METHOD PROTECTED OnExecute
hresult.Value := F_VN_MinPixelValueExp(
	ipImage := ipImage.Value,
    aMinValue := aMinValue.Value,
    aPosition := aPosition.Value,
    ipMask := ipMask.Value,
    eVectorCompareMethod := eVectorCompareMethod.Value,
	hrPrev:= hrPrev.Value);
END_METHOD

METHOD PUBLIC PreExecutionCheck
VAR_INPUT
	Check : I_PreExecutionChecks;
END_VAR
Check.IsTrue(ipImage.IsValid, 'ipImage must contain an image');
Check.IsTrue((ipImage.HasChannelCount(1) OR
              ipImage.HasChannelCount(2) OR
              ipImage.HasChannelCount(3) OR
              ipImage.HasChannelCount(4)), 'ipImage must contain 1, 2, 3 or 4 channels');

// ipMask : Optional mask to specify which pixel positions are considered (USINT, set parameter to 0 if not required)
IF NOT IsValidImage(ipMask.Value) THEN
    RETURN;
END_IF

Check.IsTrue(ipMask.IsValid, 'ipMask must contain an image');
Check.IsTrue(ipMask.HasChannelCount(1), 'ipMask must have 1 channel');
Check.IsTrue(ipMask.IsPixelDepth(8), 'ipMask must have 8 bit pixel depth');
Check.IsTrue(IsImage1SizeEqualToImage2Size(ipMask.Value, ipImage.Value), 'ipMask must be the same size as ipImage');
END_METHOD

END_FUNCTION_BLOCK

// ---- Nodes/Image Analysis/Node_F_VN_MinPixelValue.TcPOU
{attribute 'linkalways'} 
{attribute 'no_explicit_call' := 'This FB is a CLASS and must be accessed using methods or properties'}
{attribute 'enable_dynamic_creation'}
FUNCTION_BLOCK Node_F_VN_MinPixelValue EXTENDS VisionNode
VAR
    ipImage : _ITcVnImage;
    aMinValue : _TcVnVector4_LREAL;
    aPosition : _TcVnPoint2_DINT;
    hrPrev : _HRESULT(S_OK);
	hresult : _HRESULT(S_OK);
END_VAR

METHOD PUBLIC  Clone : I_Node
VAR
	pNode : POINTER TO Node_F_VN_MinPixelValue;
END_VAR
pNode := __NEW(Node_F_VN_MinPixelValue);
Clone := pNode^;
END_METHOD

METHOD FB_init : BOOL
VAR_INPUT
	bInitRetains : BOOL; // if TRUE, the retain variables are initialized (warm start / cold start)
	bInCopyCode : BOOL;  // if TRUE, the instance afterwards gets moved into the copy code (online change)
END_VAR
AddInput('ipImage', ipImage);
AddInput('hrPrev', hrPrev);
AddOutput('aMinValue', aMinValue);
AddOutput('aPosition', aPosition);
AddOutput('hresult', hresult);
END_METHOD

METHOD PROTECTED OnExecute
hresult.Value := F_VN_MinPixelValue(
	ipImage := ipImage.Value,
    aMinValue := aMinValue.Value,
    aPosition := aPosition.Value,
	hrPrev:= hrPrev.Value);
END_METHOD

METHOD PUBLIC PreExecutionCheck
VAR_INPUT
	Check : I_PreExecutionChecks;
END_VAR
Check.IsTrue(ipImage.IsValid, 'ipImage must contain an image');
Check.IsTrue((ipImage.HasChannelCount(1) OR
              ipImage.HasChannelCount(2) OR
              ipImage.HasChannelCount(3) OR
              ipImage.HasChannelCount(4)), 'ipImage must contain 1, 2, 3 or 4 channels');
END_METHOD

END_FUNCTION_BLOCK

// ---- Nodes/Image Analysis/Node_F_VN_RegionOrientationExp.TcPOU
{attribute 'linkalways'} 
{attribute 'no_explicit_call' := 'This FB is a CLASS and must be accessed using methods or properties'}
{attribute 'enable_dynamic_creation'}
FUNCTION_BLOCK Node_F_VN_RegionOrientationExp EXTENDS VisionNode
VAR
    ipSrcImage : _ITcVnImage;
    stOrientation : _TcVnRotatedRectangle;
    eMethod : _ETcVnOrientationMethod(ETcVnOrientationMethod.TCVN_OM_PCA);
    hrPrev : _HRESULT(S_OK);
	hresult : _HRESULT(S_OK);
END_VAR

METHOD PUBLIC  Clone : I_Node
VAR
	pNode : POINTER TO Node_F_VN_RegionOrientationExp;
END_VAR
pNode := __NEW(Node_F_VN_RegionOrientationExp);
Clone := pNode^;
END_METHOD

METHOD FB_init : BOOL
VAR_INPUT
	bInitRetains : BOOL; // if TRUE, the retain variables are initialized (warm start / cold start)
	bInCopyCode : BOOL;  // if TRUE, the instance afterwards gets moved into the copy code (online change)
END_VAR
AddInput('ipSrcImage', ipSrcImage);
AddParameter('eMethod', eMethod);
AddInput('hrPrev', hrPrev);
AddOutput('stOrientation', stOrientation);
AddOutput('hresult', hresult);
END_METHOD

METHOD PROTECTED OnExecute
hresult.Value := F_VN_RegionOrientationExp(
	ipSrcImage := ipSrcImage.Value,
    stOrientation := stOrientation.Value,
    eMethod := eMethod.Value,
	hrPrev:= hrPrev.Value);
END_METHOD

METHOD PUBLIC PreExecutionCheck
VAR_INPUT
	Check : I_PreExecutionChecks;
END_VAR
Check.IsTrue(ipSrcImage.IsValid, 'ipSrcImage must contain an image');
Check.IsTrue(ipSrcImage.HasChannelCount(1), 'ipSrcImage must contain 1 channel');
END_METHOD

END_FUNCTION_BLOCK

// ---- Nodes/Image Analysis/Node_F_VN_ImageAbsoluteAverage.TcPOU
{attribute 'linkalways'} 
{attribute 'no_explicit_call' := 'This FB is a CLASS and must be accessed using methods or properties'}
{attribute 'enable_dynamic_creation'}
FUNCTION_BLOCK Node_F_VN_ImageAbsoluteAverage EXTENDS VisionNode
VAR
    ipSrcImage : _ITcVnImage;
    fAverage : _LREAL(0.0);
    hrPrev : _HRESULT(S_OK);
	hresult : _HRESULT(S_OK);
END_VAR

METHOD PUBLIC  Clone : I_Node
VAR
	pNode : POINTER TO Node_F_VN_ImageAbsoluteAverage;
END_VAR
pNode := __NEW(Node_F_VN_ImageAbsoluteAverage);
Clone := pNode^;
END_METHOD

METHOD FB_init : BOOL
VAR_INPUT
	bInitRetains : BOOL; // if TRUE, the retain variables are initialized (warm start / cold start)
	bInCopyCode : BOOL;  // if TRUE, the instance afterwards gets moved into the copy code (online change)
END_VAR
AddInput('ipSrcImage', ipSrcImage);
AddInput('hrPrev', hrPrev);
AddOutput('fAverage', fAverage);
AddOutput('hresult', hresult);
END_METHOD

METHOD PROTECTED OnExecute
hresult.Value := F_VN_ImageAbsoluteAverage(
	ipSrcImage := ipSrcImage.Value,
    fAverage := fAverage.Value,
	hrPrev:= hrPrev.Value);
END_METHOD

METHOD PUBLIC PreExecutionCheck
VAR_INPUT
	Check : I_PreExecutionChecks;
END_VAR
Check.IsTrue(ipSrcImage.IsValid, 'ipSrcImage must contain an image');
END_METHOD

END_FUNCTION_BLOCK

// ---- Nodes/Image Analysis/Node_F_VN_UprightInnerRectangleExp.TcPOU
{attribute 'linkalways'} 
{attribute 'no_explicit_call' := 'This FB is a CLASS and must be accessed using methods or properties'}
{attribute 'enable_dynamic_creation'}
FUNCTION_BLOCK Node_F_VN_UprightInnerRectangleExp EXTENDS VisionNode
VAR
    ipSrcImage : _ITcVnImage;
    stRectangle : _TcVnRectangle_DINT;
    nDownScaleFactor : _DINT(-1);
    hrPrev : _HRESULT(S_OK);
	hresult : _HRESULT(S_OK);
END_VAR

METHOD PUBLIC  Clone : I_Node
VAR
	pNode : POINTER TO Node_F_VN_UprightInnerRectangleExp;
END_VAR
pNode := __NEW(Node_F_VN_UprightInnerRectangleExp);
Clone := pNode^;
END_METHOD

METHOD FB_init : BOOL
VAR_INPUT
	bInitRetains : BOOL; // if TRUE, the retain variables are initialized (warm start / cold start)
	bInCopyCode : BOOL;  // if TRUE, the instance afterwards gets moved into the copy code (online change)
END_VAR
AddInput('ipSrcImage', ipSrcImage);
AddParameter('nDownScaleFactor', nDownScaleFactor);
AddInput('hrPrev', hrPrev);
AddOutput('stRectangle', stRectangle);
AddOutput('hresult', hresult);
END_METHOD

METHOD PROTECTED OnExecute
hresult.Value := F_VN_UprightInnerRectangleExp(
	ipSrcImage := ipSrcImage.Value,
    stRectangle := stRectangle.Value,
    nDownScaleFactor := nDownScaleFactor.Value,
	hrPrev:= hrPrev.Value);
END_METHOD

METHOD PUBLIC PreExecutionCheck
VAR_INPUT
	Check : I_PreExecutionChecks;
END_VAR
Check.IsTrue(ipSrcImage.IsValid, 'ipSrcImage must contain an image');
Check.IsTrue(ipSrcImage.IsPixelDepth(8), 'ipSrcImage must be 8 bit pixel depth');
Check.IsTrue(ipSrcImage.HasChannelCount(1), 'ipSrcImage must contain 1 channel');
Check.IsTrue(nDownScaleFactor.Value >= -1, 'nDownScaleFactor must be greater than or equal to -1');
END_METHOD

END_FUNCTION_BLOCK

// ---- Nodes/Image Color and Contrast Processing/Node_F_VN_ApplyColorMap.TcPOU
{attribute 'linkalways'} 
{attribute 'no_explicit_call' := 'This FB is a CLASS and must be accessed using methods or properties'}
{attribute 'enable_dynamic_creation'}
FUNCTION_BLOCK Node_F_VN_ApplyColorMap EXTENDS VisionNode
VAR
	ipSrcImage : _ITcVnImage;
    ipDestImage : _ITcVnImage;
    ipColorMap : _ITcVnContainer;
    hrPrev : _HRESULT(S_OK);
	hresult : _HRESULT(S_OK);
END_VAR

METHOD PUBLIC  Clone : I_Node
VAR
	pNode : POINTER TO Node_F_VN_ApplyColorMap;
END_VAR
pNode := __NEW(Node_F_VN_ApplyColorMap);
Clone := pNode^;
END_METHOD

METHOD FB_init : BOOL
VAR_INPUT
	bInitRetains : BOOL; // if TRUE, the retain variables are initialized (warm start / cold start)
	bInCopyCode : BOOL;  // if TRUE, the instance afterwards gets moved into the copy code (online change)
END_VAR
AddInput('ipSrcImage', ipSrcImage);
AddInput('ipColorMap', ipColorMap);
AddInput('hrPrev', hrPrev);
AddOutput('ipDestImage', ipDestImage);
AddOutput('hresult',hresult);
END_METHOD

METHOD PROTECTED OnExecute
hresult.Value := F_VN_ApplyColorMap(
	ipSrcImage   := ipSrcImage.Value,
    ipDestImage   := ipDestImage.Value,
	ipColorMap := ipColorMap.Value,
	hrPrev := hrPrev.Value);
END_METHOD

METHOD PUBLIC PreExecutionCheck
VAR_INPUT
	Check : I_PreExecutionChecks;
END_VAR
VAR
    colorMapSize : ULINT;
END_VAR
Check.IsTrue(ipSrcImage.IsValid, 'ipSrcImage must contain an image');
Check.IsTrue(ipSrcImage.HasChannelCount(1), 'ipSrcImage must have 1 channel');

Check.IsTrue(ipColorMap.IsValid, 'ipColorMap must be a valid container');
Check.IsTrue(ipColorMap.IsType(TC_GLOBAL_CONST_LIST.ContainerType_Vector_TcVnVector3_REAL), 'ipColorMap contains incorrect type');

F_VN_GetNumberOfElements(ipColorMap.Value, colorMapSize, S_OK);

CASE colorMapSize OF
    256 :
        Check.IsTrue(ipSrcImage.IsPixelDepth(8), 'ipSrcImage must have 8 bit pixel depth');
    65536 :
        Check.IsTrue(ipSrcImage.IsPixelDepth(16), 'ipSrcImage must have 16 bit pixel depth');
ELSE
    Check.Fail('ipColorMp must contain 256 or 65536 elements');
END_CASE
END_METHOD

END_FUNCTION_BLOCK

// ---- Nodes/Image Color and Contrast Processing/Node_F_VN_Clahe.TcPOU
{attribute 'linkalways'} 
{attribute 'no_explicit_call' := 'This FB is a CLASS and must be accessed using methods or properties'}
{attribute 'enable_dynamic_creation'}
FUNCTION_BLOCK Node_F_VN_Clahe EXTENDS VisionNode
VAR
	ipSrcImage : _ITcVnImage;
    ipDestImage : _ITcVnImage;
    hrPrev : _HRESULT(S_OK);
	hresult : _HRESULT(S_OK);
END_VAR

METHOD PUBLIC  Clone : I_Node
VAR
	pNode : POINTER TO Node_F_VN_Clahe;
END_VAR
pNode := __NEW(Node_F_VN_Clahe);
Clone := pNode^;
END_METHOD

METHOD FB_init : BOOL
VAR_INPUT
	bInitRetains : BOOL; // if TRUE, the retain variables are initialized (warm start / cold start)
	bInCopyCode : BOOL;  // if TRUE, the instance afterwards gets moved into the copy code (online change)
END_VAR
AddInput('ipSrcImage', ipSrcImage);
AddInput('hrPrev', hrPrev);
AddOutput('ipDestImage', ipDestImage);
AddOutput('hresult',hresult);
END_METHOD

METHOD PROTECTED OnExecute
hresult.Value := F_VN_Clahe(
	ipSrcImage := ipSrcImage.Value,
    ipDestImage := ipDestImage.Value,
	hrPrev := hrPrev.Value);
END_METHOD

METHOD PUBLIC PreExecutionCheck
VAR_INPUT
	Check : I_PreExecutionChecks;
END_VAR
VAR
    colorMapSize : ULINT;
END_VAR
Check.IsTrue(ipSrcImage.IsValid, 'ipSrcImage must contain an image');
Check.IsTrue(ipSrcImage.HasChannelCount(1), 'ipSrcImage must have 1 channel');
Check.IsTrue((ipSrcImage.IsPixelDepth(8) OR
              ipSrcImage.IsPixelDepth(16)), 'ipSrcImage must have 8 or 16 bit pixel depth');
END_METHOD

END_FUNCTION_BLOCK

// ---- Nodes/Image Color and Contrast Processing/Node_F_VN_ClaheExp.TcPOU
{attribute 'linkalways'} 
{attribute 'no_explicit_call' := 'This FB is a CLASS and must be accessed using methods or properties'}
{attribute 'enable_dynamic_creation'}
FUNCTION_BLOCK Node_F_VN_ClaheExp EXTENDS VisionNode
VAR
	ipSrcImage : _ITcVnImage;
    ipDestImage : _ITcVnImage;
    fClipLimit  : _LREAL(0.0);
    nTilesX     : _UDINT(0);
    nTilesY     : _UDINT(0);
    hrPrev : _HRESULT(S_OK);
	hresult : _HRESULT(S_OK);
END_VAR

METHOD PUBLIC  Clone : I_Node
VAR
	pNode : POINTER TO Node_F_VN_ClaheExp;
END_VAR
pNode := __NEW(Node_F_VN_ClaheExp);
Clone := pNode^;
END_METHOD

METHOD FB_init : BOOL
VAR_INPUT
	bInitRetains : BOOL; // if TRUE, the retain variables are initialized (warm start / cold start)
	bInCopyCode : BOOL;  // if TRUE, the instance afterwards gets moved into the copy code (online change)
END_VAR
AddInput('ipSrcImage', ipSrcImage);
AddParameter('fClipLimit', fClipLimit);
AddParameter('nTilesX', nTilesX);
AddParameter('nTilesY', nTilesY);
AddInput('hrPrev', hrPrev);
AddOutput('ipDestImage', ipDestImage);
AddOutput('hresult',hresult);
END_METHOD

METHOD PROTECTED OnExecute
hresult.Value := F_VN_ClaheExp(
	ipSrcImage := ipSrcImage.Value,
    fClipLimit := fClipLimit.Value,
    nTilesX := nTilesX.Value,
    nTilesY := nTilesY.Value,
    ipDestImage   := ipDestImage.Value,
	hrPrev := hrPrev.Value);
END_METHOD

METHOD PUBLIC PreExecutionCheck
VAR_INPUT
	Check : I_PreExecutionChecks;
END_VAR
VAR
    colorMapSize : ULINT;
END_VAR
Check.IsTrue(ipSrcImage.IsValid, 'ipSrcImage must contain an image');
Check.IsTrue(ipSrcImage.HasChannelCount(1), 'ipSrcImage must have 1 channel');
Check.IsTrue((ipSrcImage.IsPixelDepth(8) OR
              ipSrcImage.IsPixelDepth(16)), 'ipSrcImage must have 8 or 16 bit pixel depth');
END_METHOD

END_FUNCTION_BLOCK

// ---- Nodes/Image Color and Contrast Processing/Node_F_VN_GenerateCustomColorMap.TcPOU
{attribute 'linkalways'} 
{attribute 'no_explicit_call' := 'This FB is a CLASS and must be accessed using methods or properties'}
{attribute 'enable_dynamic_creation'}
FUNCTION_BLOCK Node_F_VN_GenerateCustomColorMap EXTENDS VisionNode
VAR
	ipColorMap : _ITcVnContainer;
    ipInitialColors : _ITcVnContainer;
    eColorMapSize : _ETcVnColorMapSize(ETcVnColorMapSize.TCVN_CMS_256);
    hrPrev : _HRESULT(S_OK);
	hresult : _HRESULT(S_OK);
END_VAR

METHOD PUBLIC  Clone : I_Node
VAR
	pNode : POINTER TO Node_F_VN_GenerateCustomColorMap;
END_VAR
pNode := __NEW(Node_F_VN_GenerateCustomColorMap);
Clone := pNode^;
END_METHOD

METHOD FB_init : BOOL
VAR_INPUT
	bInitRetains : BOOL; // if TRUE, the retain variables are initialized (warm start / cold start)
	bInCopyCode : BOOL;  // if TRUE, the instance afterwards gets moved into the copy code (online change)
END_VAR
AddInput('ipInitialColors', ipInitialColors);
AddParameter('eColorMapSize', eColorMapSize);
AddInput('hrPrev', hrPrev);
AddOutput('ipColorMap', ipColorMap);
AddOutput('hresult',hresult);
END_METHOD

METHOD PROTECTED OnExecute
hresult.Value := F_VN_GenerateCustomColorMap(
	ipColorMap   := ipColorMap.Value,
    ipInitialColors := ipInitialColors.Value,
    eColorMapSize := eColorMapSize.Value, 
	hrPrev := hrPrev.Value);
END_METHOD

METHOD PUBLIC PreExecutionCheck
VAR_INPUT
	Check : I_PreExecutionChecks;
END_VAR
VAR
    elementNum : ULINT;
END_VAR
Check.IsTrue(ipInitialColors.IsValid, 'ipInitialColors must be a valid container');
Check.IsTrue(ipInitialColors.IsType(TC_GLOBAL_CONST_LIST.ContainerType_Vector_TcVnVector3_REAL), 'ipInitialColors contains incorrect type');
Check.IsTrue((ipInitialColors.TryGetElementNum(elementNum) AND (elementNum >= 2)), 'ipInitialColors must contain at least 2 elements');
END_METHOD

END_FUNCTION_BLOCK

// ---- Nodes/Image Color and Contrast Processing/Node_F_VN_HistogramExp.TcPOU
{attribute 'linkalways'} 
{attribute 'no_explicit_call' := 'This FB is a CLASS and must be accessed using methods or properties'}
{attribute 'enable_dynamic_creation'}
FUNCTION_BLOCK Node_F_VN_HistogramExp EXTENDS VisionNode
VAR
	ipSrcImage : _ITcVnImage;
	ipMask : _ITcVnImage;
    ipDestHistogram : _ITcVnContainer;
	nBins : _UDINT(0);
	fLowerBound : _LREAL(0.0);
	fUpperBound : _LREAL(0.0);
    hrPrev : _HRESULT(S_OK);
	hresult : _HRESULT(S_OK);
END_VAR

METHOD PUBLIC  Clone : I_Node
VAR
	pNode : POINTER TO Node_F_VN_HistogramExp;
END_VAR
pNode := __NEW(Node_F_VN_HistogramExp);
Clone := pNode^;
END_METHOD

METHOD FB_init : BOOL
VAR_INPUT
	bInitRetains : BOOL; // if TRUE, the retain variables are initialized (warm start / cold start)
	bInCopyCode : BOOL;  // if TRUE, the instance afterwards gets moved into the copy code (online change)
END_VAR
AddInput('ipSrcImage', ipSrcImage);
AddInput('ipMask', ipMask);
AddInput('hrPrev', hrPrev);
AddParameter('nBins',nBins);
AddParameter('fLowerBound',fLowerBound);
AddParameter('fUpperBound',fUpperBound);
AddOutput('ipDestHistogram', ipDestHistogram);
AddOutput('hresult',hresult);
END_METHOD

METHOD PROTECTED OnExecute
hresult.Value := F_VN_HistogramExp(
	ipSrcImage := ipSrcImage.Value,
	ipDestHistogram := ipDestHistogram.Value,
	nBins := nBins.Value,
	fLowerBound := fLowerBound.Value,
	fUpperBound := fUpperBound.Value,
	ipMask := ipMask.Value,
	hrPrev := hrPrev.Value);
END_METHOD

METHOD PUBLIC PreExecutionCheck
VAR_INPUT
	Check : I_PreExecutionChecks;
END_VAR
Check.IsTrue(ipSrcImage.IsValid, 'ipSrcImage must contain an image');
END_METHOD

END_FUNCTION_BLOCK

// ---- Nodes/Image Color and Contrast Processing/Node_F_VN_ReferenceColorSimilarity_TcVnVector3_LREAL.TcPOU
{attribute 'linkalways'} 
{attribute 'no_explicit_call' := 'This FB is a CLASS and must be accessed using methods or properties'}
{attribute 'enable_dynamic_creation'}
FUNCTION_BLOCK Node_F_VN_ReferenceColorSimilarity_TcVnVector3_LREAL EXTENDS VisionNode
VAR
	ipSrcImage : _ITcVnImage;
    ipDestImage : _ITcVnImage;
    aRefColor : _TcVnVector3_LREAL;
    hrPrev : _HRESULT(S_OK);
	hresult : _HRESULT(S_OK);
END_VAR

METHOD PUBLIC  Clone : I_Node
VAR
	pNode : POINTER TO Node_F_VN_ReferenceColorSimilarity_TcVnVector3_LREAL;
END_VAR
pNode := __NEW(Node_F_VN_ReferenceColorSimilarity_TcVnVector3_LREAL);
Clone := pNode^;
END_METHOD

METHOD FB_init : BOOL
VAR_INPUT
	bInitRetains : BOOL; // if TRUE, the retain variables are initialized (warm start / cold start)
	bInCopyCode : BOOL;  // if TRUE, the instance afterwards gets moved into the copy code (online change)
END_VAR
AddInput('ipSrcImage', ipSrcImage);
AddInput('aRefColor', aRefColor);
AddInput('hrPrev', hrPrev);
AddOutput('ipDestImage', ipDestImage);
AddOutput('hresult', hresult);
END_METHOD

METHOD PROTECTED OnExecute
hresult.Value := F_VN_ReferenceColorSimilarity_TcVnVector3_LREAL(
	ipSrcImage := ipSrcImage.Value,
    ipDestImage := ipDestImage.Value,
    aRefColor := aRefColor.Value,
	hrPrev := hrPrev.Value);
END_METHOD

METHOD PUBLIC PreExecutionCheck
VAR_INPUT
	Check : I_PreExecutionChecks;
END_VAR
VAR
    colorMapSize : ULINT;
END_VAR
Check.IsTrue(ipSrcImage.IsValid, 'ipSrcImage must contain an image');
Check.IsTrue(ipSrcImage.HasChannelCount(3), 'ipSrcImage must have 3 channels');
Check.IsTrue(ipSrcImage.IsPixelDepth(8), 'ipSrcImage must have 8 bit pixel depth');
END_METHOD

END_FUNCTION_BLOCK

// ---- Nodes/Image Color and Contrast Processing/Node_F_VN_Histogram.TcPOU
{attribute 'linkalways'} 
{attribute 'no_explicit_call' := 'This FB is a CLASS and must be accessed using methods or properties'}
{attribute 'enable_dynamic_creation'}
FUNCTION_BLOCK Node_F_VN_Histogram EXTENDS VisionNode
VAR
	ipSrcImage : _ITcVnImage;
    ipDestHistogram : _ITcVnContainer;
    hrPrev : _HRESULT(S_OK);
	hresult : _HRESULT(S_OK);
END_VAR

METHOD PUBLIC  Clone : I_Node
VAR
	pNode : POINTER TO Node_F_VN_Histogram;
END_VAR
pNode := __NEW(Node_F_VN_Histogram);
Clone := pNode^;
END_METHOD

METHOD FB_init : BOOL
VAR_INPUT
	bInitRetains : BOOL; // if TRUE, the retain variables are initialized (warm start / cold start)
	bInCopyCode : BOOL;  // if TRUE, the instance afterwards gets moved into the copy code (online change)
END_VAR
AddInput('ipSrcImage', ipSrcImage);
AddInput('hrPrev', hrPrev);
AddOutput('ipDestHistogram', ipDestHistogram);
AddOutput('hresult',hresult);
END_METHOD

METHOD PROTECTED OnExecute
hresult.Value := F_VN_Histogram(
	ipSrcImage := ipSrcImage.Value,
    ipDestHistogram := ipDestHistogram.Value,
	hrPrev := hrPrev.Value);
END_METHOD

METHOD PUBLIC PreExecutionCheck
VAR_INPUT
	Check : I_PreExecutionChecks;
END_VAR
Check.IsTrue(ipSrcImage.IsValid, 'ipSrcImage must contain an image');
END_METHOD

END_FUNCTION_BLOCK

// ---- Nodes/Image Color and Contrast Processing/Node_F_VN_HistogramEqualization.TcPOU
{attribute 'linkalways'} 
{attribute 'no_explicit_call' := 'This FB is a CLASS and must be accessed using methods or properties'}
{attribute 'enable_dynamic_creation'}
FUNCTION_BLOCK Node_F_VN_HistogramEqualization EXTENDS VisionNode
VAR
	ipSrcImage : _ITcVnImage;
    ipDestImage : _ITcVnImage;
    hrPrev : _HRESULT(S_OK);
	hresult : _HRESULT(S_OK);
END_VAR

METHOD PUBLIC  Clone : I_Node
VAR
	pNode : POINTER TO Node_F_VN_HistogramEqualization;
END_VAR
pNode := __NEW(Node_F_VN_HistogramEqualization);
Clone := pNode^;
END_METHOD

METHOD FB_init : BOOL
VAR_INPUT
	bInitRetains : BOOL; // if TRUE, the retain variables are initialized (warm start / cold start)
	bInCopyCode : BOOL;  // if TRUE, the instance afterwards gets moved into the copy code (online change)
END_VAR
AddInput('ipSrcImage', ipSrcImage);
AddInput('hrPrev', hrPrev);
AddOutput('ipDestImage', ipDestImage);
AddOutput('hresult',hresult);
END_METHOD

METHOD PROTECTED OnExecute
hresult.Value := F_VN_HistogramEqualization(
	ipSrcImage   := ipSrcImage.Value,
    ipDestImage   := ipDestImage.Value,
	hrPrev := hrPrev.Value);
END_METHOD

METHOD PUBLIC PreExecutionCheck
VAR_INPUT
	Check : I_PreExecutionChecks;
END_VAR
Check.IsTrue(ipSrcImage.IsValid, 'ipSrcImage must contain an image');
Check.IsTrue((ipSrcImage.HasChannelCount(1) OR ipSrcImage.HasChannelCount(3)), 'ipSrcImage must have 1 or 3 channels');
END_METHOD

END_FUNCTION_BLOCK

// ---- Nodes/Image Color and Contrast Processing/Node_F_VN_HistogramEqualizationExp.TcPOU
{attribute 'linkalways'} 
{attribute 'no_explicit_call' := 'This FB is a CLASS and must be accessed using methods or properties'}
{attribute 'enable_dynamic_creation'}
FUNCTION_BLOCK Node_F_VN_HistogramEqualizationExp EXTENDS VisionNode
VAR
	ipSrcImage : _ITcVnImage;
    ipDestImage : _ITcVnImage;
    hrPrev : _HRESULT(S_OK);
    nChannelIdx : _INT(-1);
	hresult : _HRESULT(S_OK);
END_VAR

METHOD PUBLIC  Clone : I_Node
VAR
	pNode : POINTER TO Node_F_VN_HistogramEqualizationExp;
END_VAR
pNode := __NEW(Node_F_VN_HistogramEqualizationExp);
Clone := pNode^;
END_METHOD

METHOD FB_init : BOOL
VAR_INPUT
	bInitRetains : BOOL; // if TRUE, the retain variables are initialized (warm start / cold start)
	bInCopyCode : BOOL;  // if TRUE, the instance afterwards gets moved into the copy code (online change)
END_VAR
AddInput('ipSrcImage', ipSrcImage);
AddParameter('nChannelIdx', nChannelIdx);
AddInput('hrPrev', hrPrev);
AddOutput('ipDestImage', ipDestImage);
AddOutput('hresult',hresult);
END_METHOD

METHOD PROTECTED OnExecute
hresult.Value := F_VN_HistogramEqualizationExp(
	ipSrcImage   := ipSrcImage.Value,
    ipDestImage   := ipDestImage.Value,
    nChannelIdx := nChannelIdx.Value,
	hrPrev := hrPrev.Value);
END_METHOD

METHOD PUBLIC PreExecutionCheck
VAR_INPUT
	Check : I_PreExecutionChecks;
END_VAR
Check.IsTrue(ipSrcImage.IsValid, 'ipSrcImage must contain an image');
Check.IsTrue(nChannelIdx.Value >= -1, 'nChannelIdx must be greater than or equal to -1');

IF nChannelIdx.Value = -1 THEN
    Check.IsTrue(ipSrcImage.HasChannelCount(3), 'ipSrcImage must have 3 channels');
ELSE
    Check.IsTrue((ipSrcImage.HasChannelCount(1) OR ipSrcImage.HasChannelCount(3)), 'ipSrcImage must have 1 or 3 channels');
END_IF
END_METHOD

END_FUNCTION_BLOCK

// ---- Nodes/Image Color and Contrast Processing/Node_F_VN_InvertImageColor.TcPOU
{attribute 'linkalways'} 
{attribute 'no_explicit_call' := 'This FB is a CLASS and must be accessed using methods or properties'}
{attribute 'enable_dynamic_creation'}
FUNCTION_BLOCK Node_F_VN_InvertImageColor EXTENDS VisionNode
VAR
    ipSrcImage : _ITcVnImage;
    ipDestImage : _ITcVnImage;
    hrPrev : _HRESULT(S_OK);
	hresult : _HRESULT(S_OK);
END_VAR

METHOD PUBLIC  Clone : I_Node
VAR
	pNode : POINTER TO Node_F_VN_InvertImageColor;
END_VAR
pNode := __NEW(Node_F_VN_InvertImageColor);
Clone := pNode^;
END_METHOD

METHOD FB_init : BOOL
VAR_INPUT
	bInitRetains : BOOL; // if TRUE, the retain variables are initialized (warm start / cold start)
	bInCopyCode : BOOL;  // if TRUE, the instance afterwards gets moved into the copy code (online change)
END_VAR
AddInput('ipSrcImage', ipSrcImage);
AddInput('hrPrev', hrPrev);
AddOutput('ipDestImage', ipDestImage);
AddOutput('hresult',hresult);
END_METHOD

METHOD PROTECTED OnExecute
hresult.Value := F_VN_InvertImageColor(
    ipSrcImage := ipSrcImage.Value,
	ipDestImage := ipDestImage.Value,
	hrPrev:= hrPrev.Value);
END_METHOD

METHOD PUBLIC PreExecutionCheck
VAR_INPUT
	Check : I_PreExecutionChecks;
END_VAR
Check.IsTrue(ipSrcImage.IsValid, 'ipSrcImage must contain an image');
END_METHOD

END_FUNCTION_BLOCK

// ---- Nodes/Image Color and Contrast Processing/Node_F_VN_ConvertColorSpace.TcPOU
{attribute 'linkalways'} 
{attribute 'no_explicit_call' := 'This FB is a CLASS and must be accessed using methods or properties'}
{attribute 'enable_dynamic_creation'}
FUNCTION_BLOCK Node_F_VN_ConvertColorSpace EXTENDS VisionNode
VAR
	ipSrcImage : _ITcVnImage;
    ipDestImage : _ITcVnImage;
    eTransform : _ETcVnColorSpaceTransform(ETcVnColorSpaceTransform.TCVN_CST_RGBA_TO_GRAY);
    hrPrev : _HRESULT(S_OK);
	hresult : _HRESULT(S_OK);
END_VAR

METHOD PUBLIC  Clone : I_Node
VAR
	pNode : POINTER TO Node_F_VN_ConvertColorSpace;
END_VAR
pNode := __NEW(Node_F_VN_ConvertColorSpace);
Clone := pNode^;
END_METHOD

METHOD FB_init : BOOL
VAR_INPUT
	bInitRetains : BOOL; // if TRUE, the retain variables are initialized (warm start / cold start)
	bInCopyCode : BOOL;  // if TRUE, the instance afterwards gets moved into the copy code (online change)
END_VAR
AddInput('ipSrcImage', ipSrcImage);
AddInput('hrPrev', hrPrev);
AddOutput('ipDestImage', ipDestImage);
AddOutput('hresult',hresult);
AddParameter('eTransform', eTransform);
END_METHOD

METHOD PROTECTED OnExecute
hresult.Value := F_VN_ConvertColorSpace(
	ipSrcImage   := ipSrcImage.Value, 
	ipDestImage:= ipDestImage.Value, 
	eTransform := eTransform.Value, 
	hrPrev := hrPrev.Value);
END_METHOD

METHOD PUBLIC PreExecutionCheck
VAR_INPUT
	Check : I_PreExecutionChecks;
END_VAR
Check.IsTrue(ipSrcImage.IsValid, 'ipSrcImage must contain an image');

CASE eTransform.Value OF
	

	ETcVnColorSpaceTransform.TCVN_CST_BGR_565_TO_RGB,
    ETcVnColorSpaceTransform.TCVN_CST_BGR_565_TO_BGR,
    ETcVnColorSpaceTransform.TCVN_CST_BGR_565_TO_RGBA,
    ETcVnColorSpaceTransform.TCVN_CST_BGR_565_TO_BGRA,
    ETcVnColorSpaceTransform.TCVN_CST_BGR_565_TO_GRAY,
    ETcVnColorSpaceTransform.TCVN_CST_BGR_555_TO_RGB,
    ETcVnColorSpaceTransform.TCVN_CST_BGR_555_TO_BGR,
    ETcVnColorSpaceTransform.TCVN_CST_BGR_555_TO_RGBA,
    ETcVnColorSpaceTransform.TCVN_CST_BGR_555_TO_BGRA,
    ETcVnColorSpaceTransform.TCVN_CST_BGR_555_TO_GRAY :

        Check.IsTrue(ipSrcImage.HasChannelCount(2), 'ipSrcImage must have 2 channels');
		Check.IsTrue(ipSrcImage.IsPixelDepth(8), 'ipSrcImage must have 8 bits per channel');
	
    // RGB, BGR (3 channels)
    ETcVnColorSpaceTransform.TCVN_CST_BGR_TO_BGRA,
    //ETcVnColorSpaceTransform.TCVN_CST_RGB_TO_RGBA, // duplicate
    ETcVnColorSpaceTransform.TCVN_CST_BGR_TO_RGBA,
    //ETcVnColorSpaceTransform.TCVN_CST_RGB_TO_BGRA, // duplicate
    ETcVnColorSpaceTransform.TCVN_CST_BGR_TO_RGB,
    //ETcVnColorSpaceTransform.TCVN_CST_RGB_TO_BGR, // duplicate
    ETcVnColorSpaceTransform.TCVN_CST_BGR_TO_GRAY,
    ETcVnColorSpaceTransform.TCVN_CST_RGB_TO_GRAY,
    ETcVnColorSpaceTransform.TCVN_CST_RGB_TO_BGR_565,
    ETcVnColorSpaceTransform.TCVN_CST_BGR_TO_BGR_565,
    ETcVnColorSpaceTransform.TCVN_CST_RGB_TO_BGR_555,
    ETcVnColorSpaceTransform.TCVN_CST_BGR_TO_BGR_555,
    ETcVnColorSpaceTransform.TCVN_CST_BGR_TO_XYZ,
    ETcVnColorSpaceTransform.TCVN_CST_RGB_TO_XYZ,
    ETcVnColorSpaceTransform.TCVN_CST_BGR_TO_YCRCB,
    ETcVnColorSpaceTransform.TCVN_CST_RGB_TO_YCRCB,
    ETcVnColorSpaceTransform.TCVN_CST_BGR_TO_HSV,
    ETcVnColorSpaceTransform.TCVN_CST_RGB_TO_HSV,
    ETcVnColorSpaceTransform.TCVN_CST_BGR_TO_LAB,
    ETcVnColorSpaceTransform.TCVN_CST_RGB_TO_LAB,
    ETcVnColorSpaceTransform.TCVN_CST_BGR_TO_LUV,
    ETcVnColorSpaceTransform.TCVN_CST_RGB_TO_LUV,
    ETcVnColorSpaceTransform.TCVN_CST_BGR_TO_HLS,
    ETcVnColorSpaceTransform.TCVN_CST_RGB_TO_HLS,
    ETcVnColorSpaceTransform.TCVN_CST_BGR_TO_HSV_FULL,
    ETcVnColorSpaceTransform.TCVN_CST_RGB_TO_HSV_FULL,
    ETcVnColorSpaceTransform.TCVN_CST_BGR_TO_HLS_FULL,
    ETcVnColorSpaceTransform.TCVN_CST_RGB_TO_HLS_FULL,
    ETcVnColorSpaceTransform.TCVN_CST_BGR_TO_YUV,
    ETcVnColorSpaceTransform.TCVN_CST_RGB_TO_YUV,
    ETcVnColorSpaceTransform.TCVN_CST_RGB_TO_YUV_420_I420,
    ETcVnColorSpaceTransform.TCVN_CST_BGR_TO_YUV_420_I420,
    //ETcVnColorSpaceTransform.TCVN_CST_RGB_TO_YUV_420_IYUV, // duplicate
    //ETcVnColorSpaceTransform.TCVN_CST_BGR_TO_YUV_420_IYUV, // duplicate
    ETcVnColorSpaceTransform.TCVN_CST_RGB_TO_YUV_420_YV12,
    ETcVnColorSpaceTransform.TCVN_CST_BGR_TO_YUV_420_YV12 :

        Check.IsTrue(ipSrcImage.HasChannelCount(3), 'ipSrcImage must have 3 channels');
    
    // RGBA, BGRA (4 channels)
    ETcVnColorSpaceTransform.TCVN_CST_BGRA_TO_BGR,
    //ETcVnColorSpaceTransform.TCVN_CST_RGBA_TO_RGB, // duplicate
    ETcVnColorSpaceTransform.TCVN_CST_BGRA_TO_RGB,
    //ETcVnColorSpaceTransform.TCVN_CST_RGBA_TO_BGR, // duplicate
    ETcVnColorSpaceTransform.TCVN_CST_BGRA_TO_RGBA,
    //ETcVnColorSpaceTransform.TCVN_CST_RGBA_TO_BGRA, // duplicate
    ETcVnColorSpaceTransform.TCVN_CST_BGRA_TO_GRAY,
    ETcVnColorSpaceTransform.TCVN_CST_RGBA_TO_GRAY,
    ETcVnColorSpaceTransform.TCVN_CST_RGBA_TO_BGR_565,
    ETcVnColorSpaceTransform.TCVN_CST_BGRA_TO_BGR_565,
    ETcVnColorSpaceTransform.TCVN_CST_RGBA_TO_BGR_555,
    ETcVnColorSpaceTransform.TCVN_CST_BGRA_TO_BGR_555,
    ETcVnColorSpaceTransform.TCVN_CST_RGBA_TO_PREMULTIPLICATED_RGBA,
    ETcVnColorSpaceTransform.TCVN_CST_RGBA_TO_YUV_420_I420,
    ETcVnColorSpaceTransform.TCVN_CST_BGRA_TO_YUV_420_I420,
    //ETcVnColorSpaceTransform.TCVN_CST_RGBA_TO_YUV_420_IYUV, // duplicate
    //ETcVnColorSpaceTransform.TCVN_CST_BGRA_TO_YUV_420_IYUV, // duplicate
    ETcVnColorSpaceTransform.TCVN_CST_RGBA_TO_YUV_420_YV12,
    ETcVnColorSpaceTransform.TCVN_CST_BGRA_TO_YUV_420_YV12 :

        Check.IsTrue(ipSrcImage.HasChannelCount(4), 'ipSrcImage must have 4 channels');
    
    // Bayer (1 channel)
    ETcVnColorSpaceTransform.TCVN_CST_BAYER_RG_TO_BGR,
    //ETcVnColorSpaceTransform.TCVN_CST_BAYER_BG_TO_RGB, // duplicate
    ETcVnColorSpaceTransform.TCVN_CST_BAYER_GR_TO_BGR,
    //ETcVnColorSpaceTransform.TCVN_CST_BAYER_GB_TO_RGB, // duplicate
    ETcVnColorSpaceTransform.TCVN_CST_BAYER_BG_TO_BGR,
    //ETcVnColorSpaceTransform.TCVN_CST_BAYER_RG_TO_RGB, // duplicate
    ETcVnColorSpaceTransform.TCVN_CST_BAYER_GB_TO_BGR,
    //ETcVnColorSpaceTransform.TCVN_CST_BAYER_GR_TO_RGB, // duplicate
    ETcVnColorSpaceTransform.TCVN_CST_BAYER_RG_TO_BGR_VNG,
    ETcVnColorSpaceTransform.TCVN_CST_BAYER_GR_TO_BGR_VNG,
    ETcVnColorSpaceTransform.TCVN_CST_BAYER_BG_TO_BGR_VNG,
    ETcVnColorSpaceTransform.TCVN_CST_BAYER_GB_TO_BGR_VNG,
    //ETcVnColorSpaceTransform.TCVN_CST_BAYER_RG_TO_RGB_VNG, // duplicate
    //ETcVnColorSpaceTransform.TCVN_CST_BAYER_GR_TO_RGB_VNG, // duplicate
    //ETcVnColorSpaceTransform.TCVN_CST_BAYER_BG_TO_RGB_VNG, // duplicate
    //ETcVnColorSpaceTransform.TCVN_CST_BAYER_GB_TO_RGB_VNG, // duplicate
    ETcVnColorSpaceTransform.TCVN_CST_BAYER_RG_TO_GRAY,
    ETcVnColorSpaceTransform.TCVN_CST_BAYER_GR_TO_GRAY,
    ETcVnColorSpaceTransform.TCVN_CST_BAYER_BG_TO_GRAY,
    ETcVnColorSpaceTransform.TCVN_CST_BAYER_GB_TO_GRAY,
    ETcVnColorSpaceTransform.TCVN_CST_BAYER_RG_TO_BGR_EA,
    ETcVnColorSpaceTransform.TCVN_CST_BAYER_GR_TO_BGR_EA,
    ETcVnColorSpaceTransform.TCVN_CST_BAYER_BG_TO_BGR_EA,
    ETcVnColorSpaceTransform.TCVN_CST_BAYER_GB_TO_BGR_EA,
    //ETcVnColorSpaceTransform.TCVN_CST_BAYER_RG_TO_RGB_EA, // duplicate
    //ETcVnColorSpaceTransform.TCVN_CST_BAYER_GR_TO_RGB_EA, // duplicate
    //ETcVnColorSpaceTransform.TCVN_CST_BAYER_BG_TO_RGB_EA, // duplicate
    //ETcVnColorSpaceTransform.TCVN_CST_BAYER_GB_TO_RGB_EA, // duplicate
    ETcVnColorSpaceTransform.TCVN_CST_BAYER_RG_TO_BGRA,
    ETcVnColorSpaceTransform.TCVN_CST_BAYER_GR_TO_BGRA,
    ETcVnColorSpaceTransform.TCVN_CST_BAYER_BG_TO_BGRA,
    ETcVnColorSpaceTransform.TCVN_CST_BAYER_GB_TO_BGRA :
    //ETcVnColorSpaceTransform.TCVN_CST_BAYER_RG_TO_RGBA, // duplicate
    //ETcVnColorSpaceTransform.TCVN_CST_BAYER_GR_TO_RGBA, // duplicate
    //ETcVnColorSpaceTransform.TCVN_CST_BAYER_BG_TO_RGBA, // duplicate
    //ETcVnColorSpaceTransform.TCVN_CST_BAYER_GB_TO_RGBA : // duplicate

        Check.IsTrue(ipSrcImage.HasChannelCount(1), 'ipSrcImage must have 1 channel');
    
    // Gray (1 channel)
    ETcVnColorSpaceTransform.TCVN_CST_GRAY_TO_BGR,
    //ETcVnColorSpaceTransform.TCVN_CST_GRAY_TO_RGB, // duplicate
    ETcVnColorSpaceTransform.TCVN_CST_GRAY_TO_BGRA,
    //ETcVnColorSpaceTransform.TCVN_CST_GRAY_TO_RGBA, // duplicate
    ETcVnColorSpaceTransform.TCVN_CST_GRAY_TO_BGR_565,
    ETcVnColorSpaceTransform.TCVN_CST_GRAY_TO_BGR_555 :

        Check.IsTrue(ipSrcImage.HasChannelCount(1), 'ipSrcImage must have 1 channel');
    
    // XYZ (3 channels)
    ETcVnColorSpaceTransform.TCVN_CST_XYZ_TO_BGR,
    ETcVnColorSpaceTransform.TCVN_CST_XYZ_TO_RGB :

        Check.IsTrue(ipSrcImage.HasChannelCount(3), 'ipSrcImage must have 3 channels');
    
    // YCrCb (3 channels)
    ETcVnColorSpaceTransform.TCVN_CST_YCRCB_TO_BGR,
    ETcVnColorSpaceTransform.TCVN_CST_YCRCB_TO_RGB :

        Check.IsTrue(ipSrcImage.HasChannelCount(3), 'ipSrcImage must have 3 channels');
    
    // HSV (3 channels)
    ETcVnColorSpaceTransform.TCVN_CST_HSV_TO_BGR,
    ETcVnColorSpaceTransform.TCVN_CST_HSV_TO_RGB,
    ETcVnColorSpaceTransform.TCVN_CST_HSV_TO_BGR_FULL,
    ETcVnColorSpaceTransform.TCVN_CST_HSV_TO_RGB_FULL :

        Check.IsTrue(ipSrcImage.HasChannelCount(3), 'ipSrcImage must have 3 channels');
    
    // LAB (3 channels)
    ETcVnColorSpaceTransform.TCVN_CST_LAB_TO_BGR,
    ETcVnColorSpaceTransform.TCVN_CST_LAB_TO_RGB,
    ETcVnColorSpaceTransform.TCVN_CST_LAB_TO_LBGR,
    ETcVnColorSpaceTransform.TCVN_CST_LAB_TO_LRGB :

        Check.IsTrue(ipSrcImage.HasChannelCount(3), 'ipSrcImage must have 3 channels');
    
    // LUV (3 channels)
    ETcVnColorSpaceTransform.TCVN_CST_LUV_TO_BGR,
    ETcVnColorSpaceTransform.TCVN_CST_LUV_TO_RGB,
    ETcVnColorSpaceTransform.TCVN_CST_LUV_TO_LBGR,
    ETcVnColorSpaceTransform.TCVN_CST_LUV_TO_LRGB :

        Check.IsTrue(ipSrcImage.HasChannelCount(3), 'ipSrcImage must have 3 channels');
    
    // HLS (3 channels)
    ETcVnColorSpaceTransform.TCVN_CST_HLS_TO_BGR,
    ETcVnColorSpaceTransform.TCVN_CST_HLS_TO_RGB,
    ETcVnColorSpaceTransform.TCVN_CST_HLS_TO_BGR_FULL,
    ETcVnColorSpaceTransform.TCVN_CST_HLS_TO_RGB_FULL :

        Check.IsTrue(ipSrcImage.HasChannelCount(3), 'ipSrcImage must have 3 channels');
    
    // LRGB, LBGR (4 channels)
    ETcVnColorSpaceTransform.TCVN_CST_LBGR_TO_LAB,
    ETcVnColorSpaceTransform.TCVN_CST_LRGB_TO_LAB,
    ETcVnColorSpaceTransform.TCVN_CST_LBGR_TO_LUV,
    ETcVnColorSpaceTransform.TCVN_CST_LRGB_TO_LUV :

        Check.IsTrue(ipSrcImage.HasChannelCount(4), 'ipSrcImage must have 4 channels');
    
    // YUV (3 channels)
    ETcVnColorSpaceTransform.TCVN_CST_YUV_TO_BGR,
    ETcVnColorSpaceTransform.TCVN_CST_YUV_TO_RGB,
    ETcVnColorSpaceTransform.TCVN_CST_YUV_420_NV12_TO_RGB,
    ETcVnColorSpaceTransform.TCVN_CST_YUV_420_NV12_TO_BGR,
    ETcVnColorSpaceTransform.TCVN_CST_YUV_420_NV21_TO_RGB,
    ETcVnColorSpaceTransform.TCVN_CST_YUV_420_NV21_TO_BGR,
    //ETcVnColorSpaceTransform.TCVN_CST_YUV_420_SP_TO_RGB, // duplicate
    //ETcVnColorSpaceTransform.TCVN_CST_YUV_420_SP_TO_BGR, // duplicate
    ETcVnColorSpaceTransform.TCVN_CST_YUV_420_NV12_TO_RGBA,
    ETcVnColorSpaceTransform.TCVN_CST_YUV_420_NV12_TO_BGRA,
    ETcVnColorSpaceTransform.TCVN_CST_YUV_420_NV21_TO_RGBA,
    ETcVnColorSpaceTransform.TCVN_CST_YUV_420_NV21_TO_BGRA,
    //ETcVnColorSpaceTransform.TCVN_CST_YUV_420_SP_TO_RGBA, // duplicate
    //ETcVnColorSpaceTransform.TCVN_CST_YUV_420_SP_TO_BGRA, // duplicate
    ETcVnColorSpaceTransform.TCVN_CST_YUV_420_YV12_TO_RGB,
    ETcVnColorSpaceTransform.TCVN_CST_YUV_420_YV12_TO_BGR,
    ETcVnColorSpaceTransform.TCVN_CST_YUV_420_IYUV_TO_RGB,
    //ETcVnColorSpaceTransform.TCVN_CST_YUV_420_I420_TO_RGB, // duplicate
    ETcVnColorSpaceTransform.TCVN_CST_YUV_420_I420_TO_BGR,
    //ETcVnColorSpaceTransform.TCVN_CST_YUV_420_P_TO_RGB, // duplicate
    //ETcVnColorSpaceTransform.TCVN_CST_YUV_420_P_TO_BGR, // duplicate
    ETcVnColorSpaceTransform.TCVN_CST_YUV_420_YV12_TO_RGBA,
    ETcVnColorSpaceTransform.TCVN_CST_YUV_420_YV12_TO_BGRA,
    ETcVnColorSpaceTransform.TCVN_CST_YUV_420_IYUV_TO_RGBA,
    ETcVnColorSpaceTransform.TCVN_CST_YUV_420_IYUV_TO_BGRA,
    //ETcVnColorSpaceTransform.TCVN_CST_YUV_420_I420_TO_RGBA, // duplicate
    //ETcVnColorSpaceTransform.TCVN_CST_YUV_420_I420_TO_BGRA, // duplicate
    //ETcVnColorSpaceTransform.TCVN_CST_YUV_420_P_TO_RGBA, // duplicate
    //ETcVnColorSpaceTransform.TCVN_CST_YUV_420_P_TO_BGRA, // duplicate
    ETcVnColorSpaceTransform.TCVN_CST_YUV_420_TO_GRAY,
    //ETcVnColorSpaceTransform.TCVN_CST_YUV_420_NV21_TO_GRAY, // duplicate
    //ETcVnColorSpaceTransform.TCVN_CST_YUV_420_NV12_TO_GRAY, // duplicate
    //ETcVnColorSpaceTransform.TCVN_CST_YUV_420_YV12_TO_GRAY, // duplicate
    //ETcVnColorSpaceTransform.TCVN_CST_YUV_420_IYUV_TO_GRAY, // duplicate
    //ETcVnColorSpaceTransform.TCVN_CST_YUV_420_I420_TO_GRAY, // duplicate
    //ETcVnColorSpaceTransform.TCVN_CST_YUV_420_SP_TO_GRAY, // duplicate
    //ETcVnColorSpaceTransform.TCVN_CST_YUV_420_P_TO_GRAY, // duplicate
    ETcVnColorSpaceTransform.TCVN_CST_YUV_422_UYVY_TO_RGB,
    ETcVnColorSpaceTransform.TCVN_CST_YUV_422_UYVY_TO_BGR,
    //ETcVnColorSpaceTransform.TCVN_CST_YUV_422_Y422_TO_RGB, // duplicate
    //ETcVnColorSpaceTransform.TCVN_CST_YUV_422_Y422_TO_BGR, // duplicate
    //ETcVnColorSpaceTransform.TCVN_CST_YUV_422_UYNV_TO_RGB, // duplicate
    //ETcVnColorSpaceTransform.TCVN_CST_YUV_422_UYNV_TO_BGR, // duplicate
    ETcVnColorSpaceTransform.TCVN_CST_YUV_422_UYVY_TO_RGBA,
    ETcVnColorSpaceTransform.TCVN_CST_YUV_422_UYVY_TO_BGRA,
    //ETcVnColorSpaceTransform.TCVN_CST_YUV_422_Y422_TO_RGBA, // duplicate
    //ETcVnColorSpaceTransform.TCVN_CST_YUV_422_Y422_TO_BGRA, // duplicate
    //ETcVnColorSpaceTransform.TCVN_CST_YUV_422_UYNV_TO_RGBA, // duplicate
    //ETcVnColorSpaceTransform.TCVN_CST_YUV_422_UYNV_TO_BGRA, // duplicate
    ETcVnColorSpaceTransform.TCVN_CST_YUV_422_YUY2_TO_RGB,
    ETcVnColorSpaceTransform.TCVN_CST_YUV_422_YUY2_TO_BGR,
    ETcVnColorSpaceTransform.TCVN_CST_YUV_422_YVYU_TO_RGB,
    ETcVnColorSpaceTransform.TCVN_CST_YUV_422_YVYU_TO_BGR,
    //ETcVnColorSpaceTransform.TCVN_CST_YUV_422_YUYV_TO_RGB, // duplicate
    //ETcVnColorSpaceTransform.TCVN_CST_YUV_422_YUYV_TO_BGR, // duplicate
    //ETcVnColorSpaceTransform.TCVN_CST_YUV_422_YUNV_TO_RGB, // duplicate
    //ETcVnColorSpaceTransform.TCVN_CST_YUV_422_YUNV_TO_BGR, // duplicate
    ETcVnColorSpaceTransform.TCVN_CST_YUV_422_YUY2_TO_RGBA,
    ETcVnColorSpaceTransform.TCVN_CST_YUV_422_YUY2_TO_BGRA,
    ETcVnColorSpaceTransform.TCVN_CST_YUV_422_YVYU_TO_RGBA,
    ETcVnColorSpaceTransform.TCVN_CST_YUV_422_YVYU_TO_BGRA,
    //ETcVnColorSpaceTransform.TCVN_CST_YUV_422_YUYV_TO_RGBA, // duplicate
    //ETcVnColorSpaceTransform.TCVN_CST_YUV_422_YUYV_TO_BGRA, // duplicate
    //ETcVnColorSpaceTransform.TCVN_CST_YUV_422_YUNV_TO_RGBA, // duplicate
    //ETcVnColorSpaceTransform.TCVN_CST_YUV_422_YUNV_TO_BGRA, // duplicate
    ETcVnColorSpaceTransform.TCVN_CST_YUV_422_UYVY_TO_GRAY,
    ETcVnColorSpaceTransform.TCVN_CST_YUV_422_YUY2_TO_GRAY :
    //ETcVnColorSpaceTransform.TCVN_CST_YUV_422_Y422_TO_GRAY, // duplicate
    //ETcVnColorSpaceTransform.TCVN_CST_YUV_422_UYNV_TO_GRAY, // duplicate
    //ETcVnColorSpaceTransform.TCVN_CST_YUV_422_YVYU_TO_GRAY, // duplicate
    //ETcVnColorSpaceTransform.TCVN_CST_YUV_422_YUYV_TO_GRAY, // duplicate
    //ETcVnColorSpaceTransform.TCVN_CST_YUV_422_YUNV_TO_GRAY : // duplicate

        Check.IsTrue(ipSrcImage.HasChannelCount(3), 'ipSrcImage must have 3 channels');
    
    // Premultiplicated RGBA (4channels)
    ETcVnColorSpaceTransform.TCVN_CST_PREMULTIPLICATED_RGBA_TO_RGBA :

        Check.IsTrue(ipSrcImage.HasChannelCount(4), 'ipSrcImage must have 4 channels');
    
    ETcVnColorSpaceTransform.TCVN_CST_MAX :

        Check.Fail('eTransform value is invalid');
ELSE
    Check.Fail('eTransform value is unknown');
END_CASE
END_METHOD

END_FUNCTION_BLOCK

// ---- Nodes/Image Color and Contrast Processing/Node_F_VN_GenerateColorMap.TcPOU
{attribute 'linkalways'} 
{attribute 'no_explicit_call' := 'This FB is a CLASS and must be accessed using methods or properties'}
{attribute 'enable_dynamic_creation'}
FUNCTION_BLOCK Node_F_VN_GenerateColorMap EXTENDS VisionNode
VAR
	ipColorMap : _ITcVnContainer;
    eColorMap : _ETcVnColorMap(ETcVnColorMap.TCVN_CM_AUTUMN);
    eColorMapSize : _ETcVnColorMapSize(ETcVnColorMapSize.TCVN_CMS_256);
    hrPrev : _HRESULT(S_OK);
	hresult : _HRESULT(S_OK);
END_VAR

METHOD PUBLIC  Clone : I_Node
VAR
	pNode : POINTER TO Node_F_VN_GenerateColorMap;
END_VAR
pNode := __NEW(Node_F_VN_GenerateColorMap);
Clone := pNode^;
END_METHOD

METHOD FB_init : BOOL
VAR_INPUT
	bInitRetains : BOOL; // if TRUE, the retain variables are initialized (warm start / cold start)
	bInCopyCode : BOOL;  // if TRUE, the instance afterwards gets moved into the copy code (online change)
END_VAR
AddParameter('eColorMap', eColorMap);
AddParameter('eColorMapSize', eColorMapSize);
AddInput('hrPrev', hrPrev);
AddOutput('ipColorMap', ipColorMap);
AddOutput('hresult', hresult);
END_METHOD

METHOD PROTECTED OnExecute
hresult.Value := F_VN_GenerateColorMap(
	ipColorMap   := ipColorMap.Value,
	eColorMap := eColorMap.Value,
    eColorMapSize := eColorMapSize.Value, 
	hrPrev := hrPrev.Value);
END_METHOD

METHOD PUBLIC PreExecutionCheck
VAR_INPUT
	Check : I_PreExecutionChecks;
END_VAR
END_METHOD

END_FUNCTION_BLOCK

// ---- Nodes/Image Color and Contrast Processing/Node_F_VN_NormalizeImage.TcPOU
{attribute 'linkalways'} 
{attribute 'no_explicit_call' := 'This FB is a CLASS and must be accessed using methods or properties'}
{attribute 'enable_dynamic_creation'}
FUNCTION_BLOCK Node_F_VN_NormalizeImage EXTENDS VisionNode
VAR
    ipSrcImage : _ITcVnImage;
    ipDestImage : _ITcVnImage;
    hrPrev : _HRESULT(S_OK);
	hresult : _HRESULT(S_OK);
END_VAR

METHOD PUBLIC  Clone : I_Node
VAR
	pNode : POINTER TO Node_F_VN_NormalizeImage;
END_VAR
pNode := __NEW(Node_F_VN_NormalizeImage);
Clone := pNode^;
END_METHOD

METHOD FB_init : BOOL
VAR_INPUT
	bInitRetains : BOOL; // if TRUE, the retain variables are initialized (warm start / cold start)
	bInCopyCode : BOOL;  // if TRUE, the instance afterwards gets moved into the copy code (online change)
END_VAR
AddInput('ipSrcImage', ipSrcImage);
AddInput('hrPrev', hrPrev);
AddOutput('ipDestImage', ipDestImage);
AddOutput('hresult',hresult);
END_METHOD

METHOD PROTECTED OnExecute
hresult.Value := F_VN_NormalizeImage(
    ipSrcImage := ipSrcImage.Value,
	ipDestImage := ipDestImage.Value,
	hrPrev:= hrPrev.Value);
END_METHOD

METHOD PUBLIC PreExecutionCheck
VAR_INPUT
	Check : I_PreExecutionChecks;
END_VAR
Check.IsTrue(ipSrcImage.IsValid, 'ipSrcImage must contain an image');
END_METHOD

END_FUNCTION_BLOCK

// ---- Nodes/Image Color and Contrast Processing/Node_F_VN_NormalizeImageForDisplay.TcPOU
{attribute 'linkalways'} 
{attribute 'no_explicit_call' := 'This FB is a CLASS and must be accessed using methods or properties'}
{attribute 'enable_dynamic_creation'}
FUNCTION_BLOCK Node_F_VN_NormalizeImageForDisplay EXTENDS VisionNode
VAR
    ipSrcImage : _ITcVnImage;
    ipDestImage : _ITcVnImage;
    eSignedNormalization : _ETcVnSignedNormalization(ETcVnSignedNormalization.TCVN_SN_FIX_ZERO);
    hrPrev : _HRESULT(S_OK);
	hresult : _HRESULT(S_OK);
END_VAR

METHOD PUBLIC  Clone : I_Node
VAR
	pNode : POINTER TO Node_F_VN_NormalizeImageForDisplay;
END_VAR
pNode := __NEW(Node_F_VN_NormalizeImageForDisplay);
Clone := pNode^;
END_METHOD

METHOD FB_init : BOOL
VAR_INPUT
	bInitRetains : BOOL; // if TRUE, the retain variables are initialized (warm start / cold start)
	bInCopyCode : BOOL;  // if TRUE, the instance afterwards gets moved into the copy code (online change)
END_VAR
AddInput('ipSrcImage', ipSrcImage);
AddInput('hrPrev', hrPrev);
AddParameter('eSignedNormalization', eSignedNormalization);
AddOutput('ipDestImage', ipDestImage);
AddOutput('hresult',hresult);
END_METHOD

METHOD PROTECTED OnExecute
hresult.Value := F_VN_NormalizeImageForDisplay(
    ipSrcImage := ipSrcImage.Value,
	ipDestImage := ipDestImage.Value,
    eSignedNormalization := eSignedNormalization.Value,
	hrPrev:= hrPrev.Value);
END_METHOD

METHOD PUBLIC PreExecutionCheck
VAR_INPUT
	Check : I_PreExecutionChecks;
END_VAR
Check.IsTrue(ipSrcImage.IsValid, 'ipSrcImage must contain an image');
END_METHOD

END_FUNCTION_BLOCK

// ---- Nodes/Image Color and Contrast Processing/Node_F_VN_ReferenceColorSimilarityExp_TcVnVector3_LREAL.TcPOU
{attribute 'linkalways'} 
{attribute 'no_explicit_call' := 'This FB is a CLASS and must be accessed using methods or properties'}
{attribute 'enable_dynamic_creation'}
FUNCTION_BLOCK Node_F_VN_ReferenceColorSimilarityExp_TcVnVector3_LREAL EXTENDS VisionNode
VAR
	ipSrcImage : _ITcVnImage;
    ipDestImage : _ITcVnImage;
    aRefColor : _TcVnVector3_LREAL;
    fVariance : _REAL(0.0);
    fLuminanceWeight : _REAL(0.0);
    hrPrev : _HRESULT(S_OK);
	hresult : _HRESULT(S_OK);
END_VAR

METHOD PUBLIC  Clone : I_Node
VAR
	pNode : POINTER TO Node_F_VN_ReferenceColorSimilarityExp_TcVnVector3_LREAL;
END_VAR
pNode := __NEW(Node_F_VN_ReferenceColorSimilarityExp_TcVnVector3_LREAL);
Clone := pNode^;
END_METHOD

METHOD FB_init : BOOL
VAR_INPUT
	bInitRetains : BOOL; // if TRUE, the retain variables are initialized (warm start / cold start)
	bInCopyCode : BOOL;  // if TRUE, the instance afterwards gets moved into the copy code (online change)
END_VAR
AddInput('ipSrcImage', ipSrcImage);
AddInput('aRefColor', aRefColor);
AddParameter('fVariance', fVariance);
AddParameter('fLuminanceWeight', fLuminanceWeight);
AddInput('hrPrev', hrPrev);
AddOutput('ipDestImage', ipDestImage);
AddOutput('hresult', hresult);
END_METHOD

METHOD PROTECTED OnExecute
hresult.Value := F_VN_ReferenceColorSimilarityExp_TcVnVector3_LREAL(
	ipSrcImage := ipSrcImage.Value,
    ipDestImage := ipDestImage.Value,
    aRefColor := aRefColor.Value,
    fVariance := fVariance.Value,
    fLuminanceWeight := fLuminanceWeight.Value,
	hrPrev := hrPrev.Value);
END_METHOD

METHOD PUBLIC PreExecutionCheck
VAR_INPUT
	Check : I_PreExecutionChecks;
END_VAR
VAR
    colorMapSize : ULINT;
END_VAR
Check.IsTrue(ipSrcImage.IsValid, 'ipSrcImage must contain an image');
Check.IsTrue(ipSrcImage.HasChannelCount(3), 'ipSrcImage must have 3 channels');
Check.IsTrue(ipSrcImage.IsPixelDepth(8), 'ipSrcImage must have 8 bit pixel depth');
Check.IsTrue(((fLuminanceWeight.Value >= 0) AND (fLuminanceWeight.Value <= 1)), 'fLuminanceWeight must be between 0 and 1');
END_METHOD

END_FUNCTION_BLOCK

// ---- Nodes/Image Color and Contrast Processing/Node_F_VN_WhiteBalance.TcPOU
{attribute 'linkalways'} 
{attribute 'no_explicit_call' := 'This FB is a CLASS and must be accessed using methods or properties'}
{attribute 'enable_dynamic_creation'}
FUNCTION_BLOCK Node_F_VN_WhiteBalance EXTENDS VisionNode
VAR
    ipSrcImage : _ITcVnImage;
    ipDestImage : _ITcVnImage;
    fRatioRed : _REAL(0);
    fRatioBlue : _REAL(0);
    nMaxValue : _UDINT(255);
    hrPrev : _HRESULT(S_OK);
	hresult : _HRESULT(S_OK);
END_VAR

METHOD PUBLIC  Clone : I_Node
VAR
	pNode : POINTER TO Node_F_VN_WhiteBalance;
END_VAR
pNode := __NEW(Node_F_VN_WhiteBalance);
Clone := pNode^;
END_METHOD

METHOD FB_init : BOOL
VAR_INPUT
	bInitRetains : BOOL; // if TRUE, the retain variables are initialized (warm start / cold start)
	bInCopyCode : BOOL;  // if TRUE, the instance afterwards gets moved into the copy code (online change)
END_VAR
AddInput('ipSrcImage', ipSrcImage);
AddInput('ipDestImage', ipDestImage);
AddParameter('nMaxValue', nMaxValue);
AddInput('hrPrev', hrPrev);
AddOutput('ipDestImage', ipDestImage);
AddOutput('fRatioRed', fRatioRed);
AddOutput('fRatioBlue', fRatioBlue);
AddOutput('hresult',hresult);
END_METHOD

METHOD PROTECTED OnExecute
hresult.Value := F_VN_WhiteBalance(
    ipSrcImage := ipSrcImage.Value,
	ipDestImage := ipDestImage.Value,
    fRatioRed := fRatioRed.Value,
    fRatioBlue := fRatioBlue.Value,
    nMaxValue := nMaxValue.Value,
	hrPrev:= hrPrev.Value);
END_METHOD

METHOD PUBLIC PreExecutionCheck
VAR_INPUT
	Check : I_PreExecutionChecks;
END_VAR
Check.IsTrue(ipSrcImage.IsValid, 'ipSrcImage must contain an image');
Check.IsTrue(ipSrcImage.HasChannelCount(3), 'ipSrcImage must have 3 channels');
Check.IsTrue((ipSrcImage.IsPixelDepth(8) OR ipSrcImage.IsPixelDepth(16)), 'ipSrcImage must have 8 or 16 bit pixel depth');
END_METHOD

END_FUNCTION_BLOCK

// ---- Nodes/Image Filtering/Node_F_VN_BilateralFilter.TcPOU
{attribute 'linkalways'} 
{attribute 'no_explicit_call' := 'This FB is a CLASS and must be accessed using methods or properties'}
{attribute 'enable_dynamic_creation'}
FUNCTION_BLOCK Node_F_VN_BilateralFilter EXTENDS VisionNode
VAR
	ipSrcImage : _ITcVnImage;
    ipDestImage : _ITcVnImage;
    nDiameter : _DINT(1);
    fSigmaColor : _LREAL(10.0);
    fSigmaSpace : _LREAL(10.0);
    hrPrev : _HRESULT(S_OK);
	hresult : _HRESULT(S_OK);
END_VAR

METHOD PUBLIC  Clone : I_Node
VAR
	pNode : POINTER TO Node_F_VN_BilateralFilter;
END_VAR
pNode := __NEW(Node_F_VN_BilateralFilter);
Clone := pNode^;
END_METHOD

METHOD FB_init : BOOL
VAR_INPUT
	bInitRetains : BOOL; // if TRUE, the retain variables are initialized (warm start / cold start)
	bInCopyCode : BOOL;  // if TRUE, the instance afterwards gets moved into the copy code (online change)
END_VAR
AddInput('ipSrcImage', ipSrcImage);
AddParameter('nDiameter', nDiameter);
AddParameter('fSigmaColor', fSigmaColor);
AddParameter('fSigmaSpace', fSigmaSpace);
AddInput('hrPrev', hrPrev);
AddOutput('ipDestImage', ipDestImage);
AddOutput('hresult',hresult);
END_METHOD

METHOD PROTECTED OnExecute
hresult.Value := F_VN_BilateralFilter(
	ipSrcImage:= ipSrcImage.Value,
	ipDestImage:= ipDestImage.Value,
	nDiameter:= nDiameter.Value,
    fSigmaColor := fSigmaColor.Value,
    fSigmaSpace := fSigmaSpace.Value,
	hrPrev:= hrPrev.Value);
END_METHOD

METHOD PUBLIC PreExecutionCheck
VAR_INPUT
	Check : I_PreExecutionChecks;
END_VAR
Check.IsTrue(ipSrcImage.IsValid, 'ipSrcImage must contain an image');
Check.IsTrue((ipSrcImage.HasChannelCount(1) OR ipSrcImage.HasChannelCount(3)), 'ipSrcImage must have 1 or 3 channels');
Check.IsTrue(ipSrcImage.IsPixelDepth(8), 'ipSrcImage must have 8 bit pixel depth');
Check.IsTrue((nDiameter.IsOdd OR nDiameter.Value = 0),'nDiameter must be odd or 0');
Check.IsTrue(fSigmaColor.Value > 0, 'fSigmaColor must be greater than 0');
Check.IsTrue(fSigmaSpace.Value > 0, 'fSigmaSpace must be greater than 0');
END_METHOD

END_FUNCTION_BLOCK

// ---- Nodes/Image Filtering/Node_F_VN_BoxFilterExp.TcPOU
{attribute 'linkalways'} 
{attribute 'no_explicit_call' := 'This FB is a CLASS and must be accessed using methods or properties'}
{attribute 'enable_dynamic_creation'}
FUNCTION_BLOCK Node_F_VN_BoxFilterExp EXTENDS VisionNode
VAR
	ipSrcImage : _ITcVnImage;
    ipDestImage : _ITcVnImage;
    nFilterWidth : _UDINT(1);
    nFilterHeight : _UDINT(1);
    eDestDepth : _ETcVnElementType(ETcVnElementType.TCVN_ET_SAME_AS_SOURCE);
    bNormalize : _BOOL(FALSE);
    eBorderType : _ETcVnBorderInterpolationMethod(ETcVnBorderInterpolationMethod.TCVN_BIM_DEFAULT);
    aAnchor : _TcVnPoint;
    hrPrev : _HRESULT(S_OK);
	hresult : _HRESULT(S_OK);
END_VAR

METHOD PUBLIC  Clone : I_Node
VAR
	pNode : POINTER TO Node_F_VN_BoxFilterExp;
END_VAR
pNode := __NEW(Node_F_VN_BoxFilterExp);
Clone := pNode^;
END_METHOD

METHOD FB_init : BOOL
VAR_INPUT
	bInitRetains : BOOL; // if TRUE, the retain variables are initialized (warm start / cold start)
	bInCopyCode : BOOL;  // if TRUE, the instance afterwards gets moved into the copy code (online change)
END_VAR
AddInput('ipSrcImage', ipSrcImage);
AddParameter('nFilterWidth', nFilterWidth);
AddParameter('nFilterHeight', nFilterHeight);
AddParameter('eDestDepth', eDestDepth);
AddParameter('bNormalize', bNormalize);
AddParameter('eBorderType', eBorderType);
AddInput('aAnchor', aAnchor);
AddInput('hrPrev', hrPrev);
AddOutput('ipDestImage', ipDestImage);
AddOutput('hresult',hresult);
END_METHOD

METHOD PROTECTED OnExecute
hresult.Value := F_VN_BoxFilterExp(
	ipSrcImage:= ipSrcImage.Value, 
	ipDestImage:= ipDestImage.Value, 
	nFilterWidth:= nFilterWidth.Value, 
	nFilterHeight:= nFilterHeight.Value,
    eDestDepth := eDestDepth.Value,
    aAnchor := aAnchor.Value,
    bNormalize := bNormalize.Value,
    eBorderType := eBorderType.Value,
	hrPrev := hrPrev.Value);
END_METHOD

METHOD PUBLIC PreExecutionCheck
VAR_INPUT
	Check : I_PreExecutionChecks;
END_VAR
Check.IsTrue(ipSrcImage.IsValid, 'ipSrcImage must contain an image');
Check.IsTrue((nFilterWidth.Value >= 1), 'nFilterWidth must be >= 1');
Check.IsTrue((nFilterHeight.Value >= 1), 'nFilterHeight must be >= 1');
END_METHOD

END_FUNCTION_BLOCK

// ---- Nodes/Image Filtering/Node_F_VN_GaussianFilterExp.TcPOU
{attribute 'linkalways'} 
{attribute 'no_explicit_call' := 'This FB is a CLASS and must be accessed using methods or properties'}
{attribute 'enable_dynamic_creation'}
FUNCTION_BLOCK Node_F_VN_GaussianFilterExp EXTENDS VisionNode
VAR
	ipSrcImage : _ITcVnImage;
    ipDestImage : _ITcVnImage;
    nFilterWidth : _UDINT(1);
    nFilterHeight : _UDINT(1);
    fSigmaX : _LREAL(0.0);
    fSigmaY : _LREAL(0.0);
    eBorderType : _ETcVnBorderInterpolationMethod(ETcVnBorderInterpolationMethod.TCVN_BIM_DEFAULT);
    hrPrev : _HRESULT(S_OK);
	hresult : _HRESULT(S_OK);
END_VAR

METHOD PUBLIC  Clone : I_Node
VAR
	pNode : POINTER TO Node_F_VN_GaussianFilterExp;
END_VAR
pNode := __NEW(Node_F_VN_GaussianFilterExp);
Clone := pNode^;
END_METHOD

METHOD FB_init : BOOL
VAR_INPUT
	bInitRetains : BOOL; // if TRUE, the retain variables are initialized (warm start / cold start)
	bInCopyCode : BOOL;  // if TRUE, the instance afterwards gets moved into the copy code (online change)
END_VAR
AddInput('ipSrcImage', ipSrcImage);
AddParameter('nFilterWidth', nFilterWidth);
AddParameter('nFilterHeight', nFilterHeight);
AddParameter('fSigmaX', fSigmaX);
AddParameter('fSigmaY', fSigmaY);
AddParameter('eBorderType', eBorderType);
AddInput('hrPrev', hrPrev);
AddOutput('ipDestImage', ipDestImage);
AddOutput('hresult',hresult);
END_METHOD

METHOD PROTECTED OnExecute
hresult.Value := F_VN_GaussianFilterExp(
	ipSrcImage := ipSrcImage.Value,
	ipDestImage := ipDestImage.Value,
	nFilterWidth := nFilterWidth.Value,
	nFilterHeight := nFilterHeight.Value,
    fSigmaX := fSigmaX.Value,
    fSigmaY := fSigmaY.Value,
    eBorderType := eBorderType.Value,
	hrPrev := hrPrev.Value);
END_METHOD

METHOD PUBLIC PreExecutionCheck
VAR_INPUT
	Check : I_PreExecutionChecks;
END_VAR
Check.IsTrue(ipSrcImage.IsValid, 'ipSrcImage must contain an image');
Check.IsTrue(nFilterWidth.IsOdd, 'nFilterWidth must be an odd number');
Check.IsTrue(nFilterHeight.IsOdd, 'nFilterHeight must be an odd number');
Check.IsTrue((fSigmaX.Value >= 0), 'fSigmaX must be greater than or equal to 0');
Check.IsTrue((fSigmaY.Value >= 0), 'fSigmaY must be greater than or equal to 0');
END_METHOD

END_FUNCTION_BLOCK

// ---- Nodes/Image Filtering/Node_F_VN_LaplacianFilterExp.TcPOU
{attribute 'linkalways'} 
{attribute 'no_explicit_call' := 'This FB is a CLASS and must be accessed using methods or properties'}
{attribute 'enable_dynamic_creation'}
FUNCTION_BLOCK Node_F_VN_LaplacianFilterExp EXTENDS VisionNode
VAR
	ipSrcImage : _ITcVnImage;
    ipDestImage : _ITcVnImage;
    eDestDepth : _ETcVnElementType(ETcVnElementType.TCVN_ET_SAME_AS_SOURCE);
    nKernelSize : _UDINT(1);
    fScale : _LREAL(1.0);
    fDelta : _LREAL(0.0);
    eBorderType : _ETcVnBorderInterpolationMethod(ETcVnBorderInterpolationMethod.TCVN_BIM_DEFAULT);
    hrPrev : _HRESULT(S_OK);
	hresult : _HRESULT(S_OK);
END_VAR

METHOD PUBLIC  Clone : I_Node
VAR
	pNode : POINTER TO Node_F_VN_LaplacianFilterExp;
END_VAR
pNode := __NEW(Node_F_VN_LaplacianFilterExp);
Clone := pNode^;
END_METHOD

METHOD FB_init : BOOL
VAR_INPUT
	bInitRetains : BOOL; // if TRUE, the retain variables are initialized (warm start / cold start)
	bInCopyCode : BOOL;  // if TRUE, the instance afterwards gets moved into the copy code (online change)
END_VAR
AddInput('ipSrcImage', ipSrcImage);
AddParameter('eDestDepth', eDestDepth);
AddParameter('nKernelSize', nKernelSize);
AddParameter('fScale', fScale);
AddParameter('fDelta', fDelta);
AddParameter('eBorderType', eBorderType);
AddInput('hrPrev', hrPrev);
AddOutput('ipDestImage', ipDestImage);
AddOutput('hresult',hresult);
END_METHOD

METHOD PROTECTED OnExecute
hresult.Value := F_VN_LaplacianFilterExp(
	ipSrcImage := ipSrcImage.Value,
	ipDestImage := ipDestImage.Value,
	eDestDepth := eDestDepth.Value,
    nKernelSize := nKernelSize.Value,
    fScale := fScale.Value,
    fDelta := fDelta.Value,
    eBorderType := eBorderType.Value,
	hrPrev := hrPrev.Value);
END_METHOD

METHOD PUBLIC PreExecutionCheck
VAR_INPUT
	Check : I_PreExecutionChecks;
END_VAR
VAR
	compatibleElementTypes_USINT : ARRAY [0..0] OF ETcVnElementType := [
		ETcVnElementType.TCVN_ET_USINT];
	
	compatibleElementTypes_UINT : ARRAY [0..1] OF ETcVnElementType := [
		ETcVnElementType.TCVN_ET_USINT,
		ETcVnElementType.TCVN_ET_UINT];
	
	compatibleElementTypes_INT : ARRAY [0..1] OF ETcVnElementType := [
		ETcVnElementType.TCVN_ET_USINT,
		ETcVnElementType.TCVN_ET_INT];
	
	compatibleElementTypes_REAL : ARRAY [0..3] OF ETcVnElementType := [
		ETcVnElementType.TCVN_ET_USINT,
		ETcVnElementType.TCVN_ET_UINT,
		ETcVnElementType.TCVN_ET_INT,
		ETcVnElementType.TCVN_ET_REAL];
	
	compatibleElementTypes_LREAL : ARRAY [0..3] OF ETcVnElementType := [
		ETcVnElementType.TCVN_ET_USINT,
		ETcVnElementType.TCVN_ET_UINT,
		ETcVnElementType.TCVN_ET_INT,
		ETcVnElementType.TCVN_ET_LREAL];
END_VAR
Check.IsTrue(ipSrcImage.IsValid, 'ipSrcImage must contain an image');

//The input image ipSrcImage may be in any available format, except for the data types SINT and DINT, which are generally not supported.

//Only the same or a larger data type than that of the input image can be used as the result depth, otherwise data would be lost.
//For example, a UINT cannot be converted to a USINT. 
//Furthermore, there are two restrictions, so that a UINT cannot be converted into an INT and a REAL cannot be converted into an LREAL.

CASE eDestDepth.Value OF
    ETcVnElementType.TCVN_ET_SINT,
    ETcVnElementType.TCVN_ET_DINT:
	    Check.Fail('ipSrcImage has unsupported pixel depth');
		RETURN;
        
	ETcVnElementType.TCVN_ET_USINT:
        Check.IsTrue(ImageHasCompatibleElementType(ipSrcImage.Value, compatibleElementTypes_USINT), 'ipSrcImage has incompatible pixel depth');
	
	ETcVnElementType.TCVN_ET_UINT:
	    Check.IsTrue(ImageHasCompatibleElementType(ipSrcImage.Value, compatibleElementTypes_UINT), 'ipSrcImage has incompatible pixel depth');
		
	ETcVnElementType.TCVN_ET_INT:
	    Check.IsTrue(ImageHasCompatibleElementType(ipSrcImage.Value, compatibleElementTypes_INT), 'ipSrcImage has incompatible pixel depth');
	
	ETcVnElementType.TCVN_ET_REAL:
	    Check.IsTrue(ImageHasCompatibleElementType(ipSrcImage.Value, compatibleElementTypes_REAL), 'ipSrcImage has incompatible pixel depth');
	
	ETcVnElementType.TCVN_ET_LREAL:
	    Check.IsTrue(ImageHasCompatibleElementType(ipSrcImage.Value, compatibleElementTypes_LREAL), 'ipSrcImage has incompatible pixel depth');
END_CASE

Check.IsTrue(nKernelSize.IsOdd, 'nKernelSize must be an odd number');
Check.IsTrue((nKernelSize.Value >= 1) AND (nKernelSize.Value <= 31), 'nKernelSize must be between 1 and 31');
END_METHOD

END_FUNCTION_BLOCK

// ---- Nodes/Image Filtering/Node_F_VN_ScharrFilter.TcPOU
{attribute 'linkalways'} 
{attribute 'no_explicit_call' := 'This FB is a CLASS and must be accessed using methods or properties'}
{attribute 'enable_dynamic_creation'}
FUNCTION_BLOCK Node_F_VN_ScharrFilter EXTENDS VisionNode
VAR
	ipSrcImage : _ITcVnImage;
    ipDestImage : _ITcVnImage;
    eDestDepth : _ETcVnElementType(ETcVnElementType.TCVN_ET_SAME_AS_SOURCE);
    eFilterDirection : _ETcVnFilterDirection(ETcVnFilterDirection.TCVN_FD_X);
    hrPrev : _HRESULT(S_OK);
	hresult : _HRESULT(S_OK);
END_VAR

METHOD PUBLIC  Clone : I_Node
VAR
	pNode : POINTER TO Node_F_VN_ScharrFilter;
END_VAR
pNode := __NEW(Node_F_VN_ScharrFilter);
Clone := pNode^;
END_METHOD

METHOD FB_init : BOOL
VAR_INPUT
	bInitRetains : BOOL; // if TRUE, the retain variables are initialized (warm start / cold start)
	bInCopyCode : BOOL;  // if TRUE, the instance afterwards gets moved into the copy code (online change)
END_VAR
AddInput('ipSrcImage', ipSrcImage);
AddParameter('eDestDepth', eDestDepth);
AddParameter('eFilterDirection', eFilterDirection);
AddInput('hrPrev', hrPrev);
AddOutput('ipDestImage', ipDestImage);
AddOutput('hresult',hresult);
END_METHOD

METHOD PROTECTED OnExecute
hresult.Value := F_VN_ScharrFilter(
	ipSrcImage:= ipSrcImage.Value,
	ipDestImage:= ipDestImage.Value,
	eDestDepth:= eDestDepth.Value,
	eFilterDirection:= eFilterDirection.Value,
	hrPrev:= hrPrev.Value);
END_METHOD

METHOD PUBLIC PreExecutionCheck
VAR_INPUT
	Check : I_PreExecutionChecks;
END_VAR
Check.IsTrue(ipSrcImage.IsValid, 'ipSrcImage must contain an image');
END_METHOD

END_FUNCTION_BLOCK

// ---- Nodes/Image Filtering/Node_F_VN_CreateStructuringElement.TcPOU
{attribute 'linkalways'} 
{attribute 'no_explicit_call' := 'This FB is a CLASS and must be accessed using methods or properties'}
{attribute 'enable_dynamic_creation'}
FUNCTION_BLOCK Node_F_VN_CreateStructuringElement EXTENDS VisionNode
VAR
	ipStructuringElement : _ITcVnImage;
    eShape : _ETcVnStructuringElementShape(ETcVnStructuringElementShape.TCVN_SES_RECTANGLE);
    nWidth : _UDINT(1);
    nHeight : _UDINT(1);
    hrPrev : _HRESULT(S_OK);
	hresult : _HRESULT(S_OK);
END_VAR

METHOD PUBLIC  Clone : I_Node
VAR
	pNode : POINTER TO Node_F_VN_CreateStructuringElement;
END_VAR
pNode := __NEW(Node_F_VN_CreateStructuringElement);
Clone := pNode^;
END_METHOD

METHOD FB_init : BOOL
VAR_INPUT
	bInitRetains : BOOL; // if TRUE, the retain variables are initialized (warm start / cold start)
	bInCopyCode : BOOL;  // if TRUE, the instance afterwards gets moved into the copy code (online change)
END_VAR
AddParameter('eShape', eShape);
AddParameter('nWidth', nWidth);
AddParameter('nHeight', nHeight);
AddInput('hrPrev', hrPrev);
AddOutput('ipStructuringElement', ipStructuringElement);
AddOutput('hresult',hresult);
END_METHOD

METHOD PROTECTED OnExecute
hresult.Value := F_VN_CreateStructuringElement(
	ipStructuringElement:= ipStructuringElement.Value, 
	eShape:= eShape.Value, 
	nWidth:= nWidth.Value, 
	nHeight:= nHeight.Value, 
	hrPrev:= hrPrev.Value);
END_METHOD

METHOD PUBLIC PreExecutionCheck
VAR_INPUT
	Check : I_PreExecutionChecks;
END_VAR
END_METHOD

END_FUNCTION_BLOCK

// ---- Nodes/Image Filtering/Node_F_VN_RemoveLocalMaxima.TcPOU
{attribute 'linkalways'} 
{attribute 'no_explicit_call' := 'This FB is a CLASS and must be accessed using methods or properties'}
{attribute 'enable_dynamic_creation'}
FUNCTION_BLOCK Node_F_VN_RemoveLocalMaxima EXTENDS VisionNode
VAR
    ipSrcImage : _ITcVnImage;
    ipDestImage : _ITcVnImage;
    fHeight : _LREAL(1.0);
    hrPrev : _HRESULT(S_OK);
	hresult : _HRESULT(S_OK);
END_VAR

METHOD PUBLIC  Clone : I_Node
VAR
	pNode : POINTER TO Node_F_VN_RemoveLocalMaxima;
END_VAR
pNode := __NEW(Node_F_VN_RemoveLocalMaxima);
Clone := pNode^;
END_METHOD

METHOD FB_init : BOOL
VAR_INPUT
	bInitRetains : BOOL; // if TRUE, the retain variables are initialized (warm start / cold start)
	bInCopyCode : BOOL;  // if TRUE, the instance afterwards gets moved into the copy code (online change)
END_VAR
AddInput('ipSrcImage', ipSrcImage);
AddParameter('fHeight', fHeight);
AddInput('hrPrev', hrPrev);
AddOutput('ipDestImage', ipDestImage);
AddOutput('hresult',hresult);
END_METHOD

METHOD PROTECTED OnExecute
hresult.Value := F_VN_RemoveLocalMaxima(
    ipSrcImage := ipSrcImage.Value,
	ipDestImage := ipDestImage.Value,
    fHeight := fHeight.Value,
	hrPrev:= hrPrev.Value);
END_METHOD

METHOD PUBLIC PreExecutionCheck
VAR_INPUT
	Check : I_PreExecutionChecks;
END_VAR
Check.IsTrue(ipSrcImage.IsValid, 'ipSrcImage must contain an image');
Check.IsTrue(ipSrcImage.HasChannelCount(1), 'ipSrcImage must have 1 channel');

Check.IsTrue((ipSrcImage.IsPixelDepth(8) OR
              ipSrcImage.IsPixelDepth(16) OR
              ipSrcImage.IsPixelDepth(32) OR
              ipSrcImage.IsPixelDepth(64)), 'ipSrcImage must have 8, 16, 32 or 64 bit pixel depth');

Check.IsTrue(fHeight.Value > 0, 'fHeight must be greater than 0');
END_METHOD

END_FUNCTION_BLOCK

// ---- Nodes/Image Filtering/Node_F_VN_MedianFilter.TcPOU
{attribute 'linkalways'} 
{attribute 'no_explicit_call' := 'This FB is a CLASS and must be accessed using methods or properties'}
{attribute 'enable_dynamic_creation'}
FUNCTION_BLOCK Node_F_VN_MedianFilter EXTENDS VisionNode
VAR
    ipSrcImage : _ITcVnImage;
    ipDestImage : _ITcVnImage;
    nFilterSize : _UDINT(3);
    hrPrev : _HRESULT(S_OK);
	hresult : _HRESULT(S_OK);
END_VAR

METHOD PUBLIC  Clone : I_Node
VAR
	pNode : POINTER TO Node_F_VN_MedianFilter;
END_VAR
pNode := __NEW(Node_F_VN_MedianFilter);
Clone := pNode^;
END_METHOD

METHOD FB_init : BOOL
VAR_INPUT
	bInitRetains : BOOL; // if TRUE, the retain variables are initialized (warm start / cold start)
	bInCopyCode : BOOL;  // if TRUE, the instance afterwards gets moved into the copy code (online change)
END_VAR
AddInput('ipSrcImage', ipSrcImage);
AddParameter('nFilterSize', nFilterSize);
AddInput('hrPrev', hrPrev);
AddOutput('ipDestImage', ipDestImage);
AddOutput('hresult',hresult);
END_METHOD

METHOD PROTECTED OnExecute
hresult.Value := F_VN_MedianFilter(
    ipSrcImage := ipSrcImage.Value,
	ipDestImage := ipDestImage.Value,
    nFilterSize := nFilterSize.Value,
	hrPrev:= hrPrev.Value);
END_METHOD

METHOD PUBLIC PreExecutionCheck
VAR_INPUT
	Check : I_PreExecutionChecks;
END_VAR
Check.IsTrue(ipSrcImage.IsValid, 'ipSrcImage must contain an image');
Check.IsTrue(nFilterSize.IsOdd, 'nFilterSize must be an odd number');
Check.IsTrue(nFilterSize.Value >= 3, 'nFilterSize must be greater than or equal to 3');

IF (nFilterSize.Value = 3) OR (nFilterSize.Value = 5) THEN
    Check.IsTrue((ipSrcImage.IsPixelDepth(8) OR
                  ipSrcImage.IsPixelDepth(16) OR
                  ipSrcImage.IsPixelDepth(32)), 'ipSrcImage must have 8, 16, or 32 bit pixel depth');
ELSE
    Check.IsTrue(ipSrcImage.IsPixelDepth(8), 'ipSrcImage must have 8 bit pixel depth');
END_IF
END_METHOD

END_FUNCTION_BLOCK

// ---- Nodes/Image Filtering/Node_F_VN_MorphologicalOperator.TcPOU
{attribute 'linkalways'} 
{attribute 'no_explicit_call' := 'This FB is a CLASS and must be accessed using methods or properties'}
{attribute 'enable_dynamic_creation'}
FUNCTION_BLOCK Node_F_VN_MorphologicalOperator EXTENDS VisionNode
VAR
	ipSrcImage : _ITcVnImage;
    ipDestImage : _ITcVnImage;
    eOperator : _ETcVnMorphologicalOperator(ETcVnMorphologicalOperator.TCVN_MO_EROSION);
    ipStructuringElement : _ITcVnImage;
    hrPrev : _HRESULT(S_OK);
	hresult : _HRESULT(S_OK);
END_VAR

METHOD PUBLIC  Clone : I_Node
VAR
	pNode : POINTER TO Node_F_VN_MorphologicalOperator;
END_VAR
pNode := __NEW(Node_F_VN_MorphologicalOperator);
Clone := pNode^;
END_METHOD

METHOD FB_init : BOOL
VAR_INPUT
	bInitRetains : BOOL; // if TRUE, the retain variables are initialized (warm start / cold start)
	bInCopyCode : BOOL;  // if TRUE, the instance afterwards gets moved into the copy code (online change)
END_VAR
AddInput('ipSrcImage', ipSrcImage);
AddParameter('eOperator', eOperator);
AddInput('ipStructuringElement', ipStructuringElement);
AddInput('hrPrev', hrPrev);
AddOutput('ipDestImage', ipDestImage);
AddOutput('hresult',hresult);
END_METHOD

METHOD PROTECTED OnExecute
hresult.Value := F_VN_MorphologicalOperator(
	ipSrcImage:= ipSrcImage.Value, 
	ipDestImage:= ipDestImage.Value, 
	eOperator:= eOperator.Value, 
	ipStructuringElement:= ipStructuringElement.Value, 
	hrPrev:= hrPrev.Value);
END_METHOD

METHOD PUBLIC PreExecutionCheck
VAR_INPUT
	Check : I_PreExecutionChecks;
END_VAR
Check.IsTrue(ipSrcImage.IsValid, 'ipSrcImage must contain an image');
Check.IsTrue(ipSrcImage.HasChannelCount(1), 'ipSrcImage must have 1 channel');
Check.IsTrue(ipStructuringElement.IsValid, 'ipStructuringElement must contain an image');
END_METHOD

END_FUNCTION_BLOCK

// ---- Nodes/Image Filtering/Node_F_VN_RemoveLocalMinima.TcPOU
{attribute 'linkalways'} 
{attribute 'no_explicit_call' := 'This FB is a CLASS and must be accessed using methods or properties'}
{attribute 'enable_dynamic_creation'}
FUNCTION_BLOCK Node_F_VN_RemoveLocalMinima EXTENDS VisionNode
VAR
    ipSrcImage : _ITcVnImage;
    ipDestImage : _ITcVnImage;
    fHeight : _LREAL(1.0);
    hrPrev : _HRESULT(S_OK);
	hresult : _HRESULT(S_OK);
END_VAR

METHOD PUBLIC  Clone : I_Node
VAR
	pNode : POINTER TO Node_F_VN_RemoveLocalMinima;
END_VAR
pNode := __NEW(Node_F_VN_RemoveLocalMinima);
Clone := pNode^;
END_METHOD

METHOD FB_init : BOOL
VAR_INPUT
	bInitRetains : BOOL; // if TRUE, the retain variables are initialized (warm start / cold start)
	bInCopyCode : BOOL;  // if TRUE, the instance afterwards gets moved into the copy code (online change)
END_VAR
AddInput('ipSrcImage', ipSrcImage);
AddParameter('fHeight', fHeight);
AddInput('hrPrev', hrPrev);
AddOutput('ipDestImage', ipDestImage);
AddOutput('hresult',hresult);
END_METHOD

METHOD PROTECTED OnExecute
hresult.Value := F_VN_RemoveLocalMinima(
    ipSrcImage := ipSrcImage.Value,
	ipDestImage := ipDestImage.Value,
    fHeight := fHeight.Value,
	hrPrev:= hrPrev.Value);
END_METHOD

METHOD PUBLIC PreExecutionCheck
VAR_INPUT
	Check : I_PreExecutionChecks;
END_VAR
Check.IsTrue(ipSrcImage.IsValid, 'ipSrcImage must contain an image');
Check.IsTrue(ipSrcImage.HasChannelCount(1), 'ipSrcImage must have 1 channel');

Check.IsTrue((ipSrcImage.IsPixelDepth(8) OR
              ipSrcImage.IsPixelDepth(16) OR
              ipSrcImage.IsPixelDepth(32) OR
              ipSrcImage.IsPixelDepth(64)), 'ipSrcImage must have 8, 16, 32 or 64 bit pixel depth');

Check.IsTrue(fHeight.Value > 0, 'fHeight must be greater than 0');
END_METHOD

END_FUNCTION_BLOCK

// ---- Nodes/Image Filtering/Node_F_VN_ScharrFilterExp.TcPOU
{attribute 'linkalways'} 
{attribute 'no_explicit_call' := 'This FB is a CLASS and must be accessed using methods or properties'}
{attribute 'enable_dynamic_creation'}
FUNCTION_BLOCK Node_F_VN_ScharrFilterExp EXTENDS VisionNode
VAR
	ipSrcImage : _ITcVnImage;
    ipDestImage : _ITcVnImage;
    eDestDepth : _ETcVnElementType(ETcVnElementType.TCVN_ET_SAME_AS_SOURCE);
    eFilterDirection : _ETcVnFilterDirection(ETcVnFilterDirection.TCVN_FD_X);
    fScale : _LREAL(1.0);
    fDelta : _LREAL(0.0);
    eBorderType : _ETcVnBorderInterpolationMethod(ETcVnBorderInterpolationMethod.TCVN_BIM_DEFAULT);
    hrPrev : _HRESULT(S_OK);
	hresult : _HRESULT(S_OK);
END_VAR

METHOD PUBLIC  Clone : I_Node
VAR
	pNode : POINTER TO Node_F_VN_ScharrFilterExp;
END_VAR
pNode := __NEW(Node_F_VN_ScharrFilterExp);
Clone := pNode^;
END_METHOD

METHOD FB_init : BOOL
VAR_INPUT
	bInitRetains : BOOL; // if TRUE, the retain variables are initialized (warm start / cold start)
	bInCopyCode : BOOL;  // if TRUE, the instance afterwards gets moved into the copy code (online change)
END_VAR
AddInput('ipSrcImage', ipSrcImage);
AddParameter('eDestDepth', eDestDepth);
AddParameter('eFilterDirection', eFilterDirection);
AddParameter('fScale', fScale);
AddParameter('fDelta', fDelta);
AddParameter('eBorderType', eBorderType);
AddInput('hrPrev', hrPrev);
AddOutput('ipDestImage', ipDestImage);
AddOutput('hresult',hresult);
END_METHOD

METHOD PROTECTED OnExecute
hresult.Value := F_VN_ScharrFilterExp(
	ipSrcImage:= ipSrcImage.Value,
	ipDestImage:= ipDestImage.Value,
	eDestDepth:= eDestDepth.Value,
	eFilterDirection:= eFilterDirection.Value,
    fScale := fScale.Value,
    fDelta := fDelta.Value,
    eBorderType := eBorderType.Value,
	hrPrev:= hrPrev.Value);
END_METHOD

METHOD PUBLIC PreExecutionCheck
VAR_INPUT
	Check : I_PreExecutionChecks;
END_VAR
Check.IsTrue(ipSrcImage.IsValid, 'ipSrcImage must contain an image');
END_METHOD

END_FUNCTION_BLOCK

// ---- Nodes/Image Filtering/Node_F_VN_BilateralFilterExp.TcPOU
{attribute 'linkalways'} 
{attribute 'no_explicit_call' := 'This FB is a CLASS and must be accessed using methods or properties'}
{attribute 'enable_dynamic_creation'}
FUNCTION_BLOCK Node_F_VN_BilateralFilterExp EXTENDS VisionNode
VAR
	ipSrcImage : _ITcVnImage;
    ipDestImage : _ITcVnImage;
    nDiameter : _DINT(1);
    fSigmaColor : _LREAL(10.0);
    fSigmaSpace : _LREAL(10.0);
    eBorderType : _ETcVnBorderInterpolationMethod(ETcVnBorderInterpolationMethod.TCVN_BIM_DEFAULT);
    hrPrev : _HRESULT(S_OK);
	hresult : _HRESULT(S_OK);
END_VAR

METHOD PUBLIC  Clone : I_Node
VAR
	pNode : POINTER TO Node_F_VN_BilateralFilterExp;
END_VAR
pNode := __NEW(Node_F_VN_BilateralFilterExp);
Clone := pNode^;
END_METHOD

METHOD FB_init : BOOL
VAR_INPUT
	bInitRetains : BOOL; // if TRUE, the retain variables are initialized (warm start / cold start)
	bInCopyCode : BOOL;  // if TRUE, the instance afterwards gets moved into the copy code (online change)
END_VAR
AddInput('ipSrcImage', ipSrcImage);
AddParameter('nDiameter', nDiameter);
AddParameter('fSigmaColor', fSigmaColor);
AddParameter('fSigmaSpace', fSigmaSpace);
AddParameter('eBorderType', eBorderType);
AddInput('hrPrev', hrPrev);
AddOutput('ipDestImage', ipDestImage);
AddOutput('hresult',hresult);
END_METHOD

METHOD PROTECTED OnExecute
hresult.Value := F_VN_BilateralFilterExp(
	ipSrcImage:= ipSrcImage.Value,
	ipDestImage:= ipDestImage.Value,
	nDiameter:= nDiameter.Value,
    fSigmaColor := fSigmaColor.Value,
    fSigmaSpace := fSigmaSpace.Value,
    eBorderType := eBorderType.Value,
	hrPrev:= hrPrev.Value);
END_METHOD

METHOD PUBLIC PreExecutionCheck
VAR_INPUT
	Check : I_PreExecutionChecks;
END_VAR
Check.IsTrue(ipSrcImage.IsValid, 'ipSrcImage must contain an image');
Check.IsTrue((ipSrcImage.HasChannelCount(1) OR ipSrcImage.HasChannelCount(3)), 'ipSrcImage must have 1 or 3 channels');
Check.IsTrue(ipSrcImage.IsPixelDepth(8), 'ipSrcImage must have 8 bit pixel depth');
Check.IsTrue((nDiameter.IsOdd OR nDiameter.Value = 0),'nDiameter must be odd or 0');
Check.IsTrue(fSigmaColor.Value > 0, 'fSigmaColor must be greater than 0');
Check.IsTrue(fSigmaSpace.Value > 0, 'fSigmaSpace must be greater than 0');
END_METHOD

END_FUNCTION_BLOCK

// ---- Nodes/Image Filtering/Node_F_VN_SobelFilterExp.TcPOU
{attribute 'linkalways'} 
{attribute 'no_explicit_call' := 'This FB is a CLASS and must be accessed using methods or properties'}
{attribute 'enable_dynamic_creation'}
FUNCTION_BLOCK Node_F_VN_SobelFilterExp EXTENDS VisionNode
VAR
	ipSrcImage : _ITcVnImage;
    ipDestImage : _ITcVnImage;
    eDestDepth : _ETcVnElementType(ETcVnElementType.TCVN_ET_SAME_AS_SOURCE);
    nXOrder : _UDINT(0);
    nYOrder : _UDINT(0);
    nKernelSize : _UDINT(3);
    fScale : _LREAL(1.0);
    fDelta : _LREAL(0.0);
    eBorderType : _ETcVnBorderInterpolationMethod(ETcVnBorderInterpolationMethod.TCVN_BIM_DEFAULT);
    hrPrev : _HRESULT(S_OK);
	hresult : _HRESULT(S_OK);
END_VAR

METHOD PUBLIC  Clone : I_Node
VAR
	pNode : POINTER TO Node_F_VN_SobelFilterExp;
END_VAR
pNode := __NEW(Node_F_VN_SobelFilterExp);
Clone := pNode^;
END_METHOD

METHOD FB_init : BOOL
VAR_INPUT
	bInitRetains : BOOL; // if TRUE, the retain variables are initialized (warm start / cold start)
	bInCopyCode : BOOL;  // if TRUE, the instance afterwards gets moved into the copy code (online change)
END_VAR
AddInput('ipSrcImage', ipSrcImage);
AddParameter('eDestDepth', eDestDepth);
AddParameter('nXOrder', nXOrder);
AddParameter('nYOrder', nYOrder);
AddParameter('nKernelSize', nKernelSize);
AddParameter('fScale', fScale);
AddParameter('fDelta', fDelta);
AddParameter('eBorderType', eBorderType);
AddInput('hrPrev', hrPrev);
AddOutput('ipDestImage', ipDestImage);
AddOutput('hresult',hresult);
END_METHOD

METHOD PROTECTED OnExecute
hresult.Value := F_VN_SobelFilterExp(
	ipSrcImage:= ipSrcImage.Value,
	ipDestImage:= ipDestImage.Value,
	eDestDepth:= eDestDepth.Value,
	nXOrder:= nXOrder.Value,
    nYOrder:= nYOrder.Value,
    nKernelSize:= nKernelSize.Value,
    fScale := fScale.Value,
    fDelta := fDelta.Value,
    eBorderType := eBorderType.Value,
	hrPrev:= hrPrev.Value);
END_METHOD

METHOD PUBLIC PreExecutionCheck
VAR_INPUT
	Check : I_PreExecutionChecks;
END_VAR
VAR
    x_plus_y : UDINT;
END_VAR
Check.IsTrue(ipSrcImage.IsValid, 'ipSrcImage must contain an image');
Check.IsTrue(nKernelSize.IsOdd, 'nKernelSize must be an odd number');
Check.IsTrue((nKernelSize.Value >= 3), 'nKernelSize must be greater than or equal to 3');
Check.IsTrue((nKernelSize.Value <= 31), 'nKernelSize must be less than or equal to 31');

x_plus_y := nXOrder.Value + nYOrder.Value;
Check.IsTrue((x_plus_y > 0), 'nXOrder and nYOrder cannot both be 0');
Check.IsTrue((x_plus_y < nKernelSize.Value), 'nXOrder + nYOrder must be less than nKernelSize');
END_METHOD

END_FUNCTION_BLOCK

// ---- Nodes/Image Filtering/Node_F_VN_SobelFilter.TcPOU
{attribute 'linkalways'} 
{attribute 'no_explicit_call' := 'This FB is a CLASS and must be accessed using methods or properties'}
{attribute 'enable_dynamic_creation'}
FUNCTION_BLOCK Node_F_VN_SobelFilter EXTENDS VisionNode
VAR
	ipSrcImage : _ITcVnImage;
    ipDestImage : _ITcVnImage;
    eDestDepth : _ETcVnElementType(ETcVnElementType.TCVN_ET_SAME_AS_SOURCE);
    nXOrder : _UDINT(0);
    nYOrder : _UDINT(0);
    hrPrev : _HRESULT(S_OK);
	hresult : _HRESULT(S_OK);
END_VAR

METHOD PUBLIC  Clone : I_Node
VAR
	pNode : POINTER TO Node_F_VN_SobelFilter;
END_VAR
pNode := __NEW(Node_F_VN_SobelFilter);
Clone := pNode^;
END_METHOD

METHOD FB_init : BOOL
VAR_INPUT
	bInitRetains : BOOL; // if TRUE, the retain variables are initialized (warm start / cold start)
	bInCopyCode : BOOL;  // if TRUE, the instance afterwards gets moved into the copy code (online change)
END_VAR
AddInput('ipSrcImage', ipSrcImage);
AddParameter('eDestDepth', eDestDepth);
AddParameter('nXOrder', nXOrder);
AddParameter('nYOrder', nYOrder);
AddInput('hrPrev', hrPrev);
AddOutput('ipDestImage', ipDestImage);
AddOutput('hresult',hresult);
END_METHOD

METHOD PROTECTED OnExecute
hresult.Value := F_VN_SobelFilter(
	ipSrcImage:= ipSrcImage.Value,
	ipDestImage:= ipDestImage.Value,
	eDestDepth:= eDestDepth.Value,
	nXOrder:= nXOrder.Value,
    nYOrder:= nYOrder.Value,
	hrPrev:= hrPrev.Value);
END_METHOD

METHOD PUBLIC PreExecutionCheck
VAR_INPUT
	Check : I_PreExecutionChecks;
END_VAR
VAR
    x_plus_y : UDINT;
END_VAR
Check.IsTrue(ipSrcImage.IsValid, 'ipSrcImage must contain an image');

x_plus_y := nXOrder.Value + nYOrder.Value;
Check.IsTrue((x_plus_y > 0), 'nXOrder and nYOrder cannot both be 0');
Check.IsTrue((x_plus_y < 3), 'nXOrder + nYOrder must be less than 3'); // Basic SobelFilter uses a fixed kernel size of 3.
END_METHOD

END_FUNCTION_BLOCK

// ---- Nodes/Image Filtering/Node_F_VN_VarianceFilter.TcPOU
{attribute 'linkalways'} 
{attribute 'no_explicit_call' := 'This FB is a CLASS and must be accessed using methods or properties'}
{attribute 'enable_dynamic_creation'}
FUNCTION_BLOCK Node_F_VN_VarianceFilter EXTENDS VisionNode
VAR
    ipSrcImage : _ITcVnImage;
    ipDestImage : _ITcVnImage;
    nKernelSize : _UDINT(0);
    hrPrev : _HRESULT(S_OK);
	hresult : _HRESULT(S_OK);
END_VAR

METHOD PUBLIC  Clone : I_Node
VAR
	pNode : POINTER TO Node_F_VN_VarianceFilter;
END_VAR
pNode := __NEW(Node_F_VN_VarianceFilter);
Clone := pNode^;
END_METHOD

METHOD FB_init : BOOL
VAR_INPUT
	bInitRetains : BOOL; // if TRUE, the retain variables are initialized (warm start / cold start)
	bInCopyCode : BOOL;  // if TRUE, the instance afterwards gets moved into the copy code (online change)
END_VAR
AddInput('ipSrcImage', ipSrcImage);
AddParameter('nKernelSize', nKernelSize);
AddInput('hrPrev', hrPrev);
AddOutput('ipDestImage', ipDestImage);
AddOutput('hresult',hresult);
END_METHOD

METHOD PROTECTED OnExecute
hresult.Value := F_VN_VarianceFilter(
    ipSrcImage := ipSrcImage.Value,
	ipDestImage := ipDestImage.Value,
    nKernelSize := nKernelSize.Value,
	hrPrev:= hrPrev.Value);
END_METHOD

METHOD PUBLIC PreExecutionCheck
VAR_INPUT
	Check : I_PreExecutionChecks;
END_VAR
Check.IsTrue(ipSrcImage.IsValid, 'ipSrcImage must contain an image');
Check.IsTrue(ipSrcImage.HasChannelCount(1), 'ipSrcImage must have 1 channel');
Check.IsTrue(ipSrcImage.IsPixelDepth(8), 'ipSrcImage must have 8 bit pixel depth');
END_METHOD

END_FUNCTION_BLOCK

// ---- Nodes/Image Filtering/Node_F_VN_LocalMaxima.TcPOU
{attribute 'linkalways'} 
{attribute 'no_explicit_call' := 'This FB is a CLASS and must be accessed using methods or properties'}
{attribute 'enable_dynamic_creation'}
FUNCTION_BLOCK Node_F_VN_LocalMaxima EXTENDS VisionNode
VAR
    ipSrcImage : _ITcVnImage;
    ipDestImage : _ITcVnImage;
    hrPrev : _HRESULT(S_OK);
	hresult : _HRESULT(S_OK);
END_VAR

METHOD PUBLIC  Clone : I_Node
VAR
	pNode : POINTER TO Node_F_VN_LocalMaxima;
END_VAR
pNode := __NEW(Node_F_VN_LocalMaxima);
Clone := pNode^;
END_METHOD

METHOD FB_init : BOOL
VAR_INPUT
	bInitRetains : BOOL; // if TRUE, the retain variables are initialized (warm start / cold start)
	bInCopyCode : BOOL;  // if TRUE, the instance afterwards gets moved into the copy code (online change)
END_VAR
AddInput('ipSrcImage', ipSrcImage);
AddInput('hrPrev', hrPrev);
AddOutput('ipDestImage', ipDestImage);
AddOutput('hresult',hresult);
END_METHOD

METHOD PROTECTED OnExecute
hresult.Value := F_VN_LocalMaxima(
    ipSrcImage := ipSrcImage.Value,
	ipDestImage := ipDestImage.Value,
	hrPrev:= hrPrev.Value);
END_METHOD

METHOD PUBLIC PreExecutionCheck
VAR_INPUT
	Check : I_PreExecutionChecks;
END_VAR
Check.IsTrue(ipSrcImage.IsValid, 'ipSrcImage must contain an image');
Check.IsTrue(ipSrcImage.HasChannelCount(1), 'ipSrcImage must have 1 channel');

Check.IsTrue((ipSrcImage.IsPixelDepth(8)  OR
              ipSrcImage.IsPixelDepth(16)), 'ipSrcImage must have 8 or 16 bit pixel depth');
END_METHOD

END_FUNCTION_BLOCK

// ---- Nodes/Image Filtering/Node_F_VN_DarkBorderObjects.TcPOU
{attribute 'linkalways'} 
{attribute 'no_explicit_call' := 'This FB is a CLASS and must be accessed using methods or properties'}
{attribute 'enable_dynamic_creation'}
FUNCTION_BLOCK Node_F_VN_DarkBorderObjects EXTENDS VisionNode
VAR
    ipSrcImage : _ITcVnImage;
    ipDestImage : _ITcVnImage;
    hrPrev : _HRESULT(S_OK);
	hresult : _HRESULT(S_OK);
END_VAR

METHOD PUBLIC  Clone : I_Node
VAR
	pNode : POINTER TO Node_F_VN_DarkBorderObjects;
END_VAR
pNode := __NEW(Node_F_VN_DarkBorderObjects);
Clone := pNode^;
END_METHOD

METHOD FB_init : BOOL
VAR_INPUT
	bInitRetains : BOOL; // if TRUE, the retain variables are initialized (warm start / cold start)
	bInCopyCode : BOOL;  // if TRUE, the instance afterwards gets moved into the copy code (online change)
END_VAR
AddInput('ipSrcImage', ipSrcImage);
AddInput('hrPrev', hrPrev);
AddOutput('ipDestImage', ipDestImage);
AddOutput('hresult',hresult);
END_METHOD

METHOD PROTECTED OnExecute
hresult.Value := F_VN_DarkBorderObjects(
    ipSrcImage := ipSrcImage.Value,
	ipDestImage := ipDestImage.Value,
	hrPrev:= hrPrev.Value);
END_METHOD

METHOD PUBLIC PreExecutionCheck
VAR_INPUT
	Check : I_PreExecutionChecks;
END_VAR
Check.IsTrue(ipSrcImage.IsValid, 'ipSrcImage must contain an image');
Check.IsTrue(ipSrcImage.HasChannelCount(1), 'ipSrcImage must have 1 channel');

Check.IsTrue((ipSrcImage.IsPixelDepth(8)  OR
              ipSrcImage.IsPixelDepth(16) OR
              ipSrcImage.IsPixelDepth(32) OR
              ipSrcImage.IsPixelDepth(64)), 'ipSrcImage must have 8, 16, 32 or 64 bit pixel depth');
END_METHOD

END_FUNCTION_BLOCK

// ---- Nodes/Image Filtering/Node_F_VN_FillHoles.TcPOU
{attribute 'linkalways'} 
{attribute 'no_explicit_call' := 'This FB is a CLASS and must be accessed using methods or properties'}
{attribute 'enable_dynamic_creation'}
FUNCTION_BLOCK Node_F_VN_FillHoles EXTENDS VisionNode
VAR
    ipSrcImage : _ITcVnImage;
    ipDestImage : _ITcVnImage;
    hrPrev : _HRESULT(S_OK);
	hresult : _HRESULT(S_OK);
END_VAR

METHOD PUBLIC  Clone : I_Node
VAR
	pNode : POINTER TO Node_F_VN_FillHoles;
END_VAR
pNode := __NEW(Node_F_VN_FillHoles);
Clone := pNode^;
END_METHOD

METHOD FB_init : BOOL
VAR_INPUT
	bInitRetains : BOOL; // if TRUE, the retain variables are initialized (warm start / cold start)
	bInCopyCode : BOOL;  // if TRUE, the instance afterwards gets moved into the copy code (online change)
END_VAR
AddInput('ipSrcImage', ipSrcImage);
AddInput('hrPrev', hrPrev);
AddOutput('ipDestImage', ipDestImage);
AddOutput('hresult',hresult);
END_METHOD

METHOD PROTECTED OnExecute
hresult.Value := F_VN_FillHoles(
    ipSrcImage := ipSrcImage.Value,
	ipDestImage := ipDestImage.Value,
	hrPrev:= hrPrev.Value);
END_METHOD

METHOD PUBLIC PreExecutionCheck
VAR_INPUT
	Check : I_PreExecutionChecks;
END_VAR
Check.IsTrue(ipSrcImage.IsValid, 'ipSrcImage must contain an image');
Check.IsTrue(ipSrcImage.HasChannelCount(1), 'ipSrcImage must have 1 channel');

Check.IsTrue((ipSrcImage.IsPixelDepth(8)  OR
              ipSrcImage.IsPixelDepth(16) OR
              ipSrcImage.IsPixelDepth(32) OR
              ipSrcImage.IsPixelDepth(64)), 'ipSrcImage must have 8, 16, 32 or 64 bit pixel depth');
END_METHOD

END_FUNCTION_BLOCK

// ---- Nodes/Image Filtering/Node_F_VN_BoxFilter.TcPOU
{attribute 'linkalways'} 
{attribute 'no_explicit_call' := 'This FB is a CLASS and must be accessed using methods or properties'}
{attribute 'enable_dynamic_creation'}
FUNCTION_BLOCK Node_F_VN_BoxFilter EXTENDS VisionNode
VAR
	ipSrcImage : _ITcVnImage;
    ipDestImage : _ITcVnImage;
    nFilterWidth : _UDINT(1);
    nFilterHeight : _UDINT(1);
    hrPrev : _HRESULT(S_OK);
	hresult : _HRESULT(S_OK);
END_VAR

METHOD PUBLIC  Clone : I_Node
VAR
	pNode : POINTER TO Node_F_VN_BoxFilter;
END_VAR
pNode := __NEW(Node_F_VN_BoxFilter);
Clone := pNode^;
END_METHOD

METHOD FB_init : BOOL
VAR_INPUT
	bInitRetains : BOOL; // if TRUE, the retain variables are initialized (warm start / cold start)
	bInCopyCode : BOOL;  // if TRUE, the instance afterwards gets moved into the copy code (online change)
END_VAR
AddInput('ipSrcImage', ipSrcImage);
AddParameter('nFilterWidth', nFilterWidth);
AddParameter('nFilterHeight', nFilterHeight);
AddInput('hrPrev', hrPrev);
AddOutput('ipDestImage', ipDestImage);
AddOutput('hresult',hresult);
END_METHOD

METHOD PROTECTED OnExecute
hresult.Value := F_VN_BoxFilter(
	ipSrcImage:= ipSrcImage.Value, 
	ipDestImage:= ipDestImage.Value, 
	nFilterWidth:= nFilterWidth.Value, 
	nFilterHeight:= nFilterHeight.Value, 
	hrPrev:= hrPrev.Value);
END_METHOD

METHOD PUBLIC PreExecutionCheck
VAR_INPUT
	Check : I_PreExecutionChecks;
END_VAR
Check.IsTrue(ipSrcImage.IsValid, 'ipSrcImage must contain an image');
Check.IsTrue((nFilterWidth.Value >= 1), 'nFilterWidth must be >= 1');
Check.IsTrue((nFilterHeight.Value >= 1), 'nFilterHeight must be >= 1');
END_METHOD

END_FUNCTION_BLOCK

// ---- Nodes/Image Filtering/Node_F_VN_BrightBorderObjects.TcPOU
{attribute 'linkalways'} 
{attribute 'no_explicit_call' := 'This FB is a CLASS and must be accessed using methods or properties'}
{attribute 'enable_dynamic_creation'}
FUNCTION_BLOCK Node_F_VN_BrightBorderObjects EXTENDS VisionNode
VAR
    ipSrcImage : _ITcVnImage;
    ipDestImage : _ITcVnImage;
    hrPrev : _HRESULT(S_OK);
	hresult : _HRESULT(S_OK);
END_VAR

METHOD PUBLIC  Clone : I_Node
VAR
	pNode : POINTER TO Node_F_VN_BrightBorderObjects;
END_VAR
pNode := __NEW(Node_F_VN_BrightBorderObjects);
Clone := pNode^;
END_METHOD

METHOD FB_init : BOOL
VAR_INPUT
	bInitRetains : BOOL; // if TRUE, the retain variables are initialized (warm start / cold start)
	bInCopyCode : BOOL;  // if TRUE, the instance afterwards gets moved into the copy code (online change)
END_VAR
AddInput('ipSrcImage', ipSrcImage);
AddInput('hrPrev', hrPrev);
AddOutput('ipDestImage', ipDestImage);
AddOutput('hresult',hresult);
END_METHOD

METHOD PROTECTED OnExecute
hresult.Value := F_VN_BrightBorderObjects(
    ipSrcImage := ipSrcImage.Value,
	ipDestImage := ipDestImage.Value,
	hrPrev:= hrPrev.Value);
END_METHOD

METHOD PUBLIC PreExecutionCheck
VAR_INPUT
	Check : I_PreExecutionChecks;
END_VAR
Check.IsTrue(ipSrcImage.IsValid, 'ipSrcImage must contain an image');
Check.IsTrue(ipSrcImage.HasChannelCount(1), 'ipSrcImage must have 1 channel');

Check.IsTrue((ipSrcImage.IsPixelDepth(8)  OR
              ipSrcImage.IsPixelDepth(16) OR
              ipSrcImage.IsPixelDepth(32) OR
              ipSrcImage.IsPixelDepth(64)), 'ipSrcImage must have 8, 16, 32 or 64 bit pixel depth');
END_METHOD

END_FUNCTION_BLOCK

// ---- Nodes/Image Filtering/Node_F_VN_GaussianFilter.TcPOU
{attribute 'linkalways'} 
{attribute 'no_explicit_call' := 'This FB is a CLASS and must be accessed using methods or properties'}
{attribute 'enable_dynamic_creation'}
FUNCTION_BLOCK Node_F_VN_GaussianFilter EXTENDS VisionNode
VAR
	ipSrcImage : _ITcVnImage;
    ipDestImage : _ITcVnImage;
    nFilterWidth : _UDINT(1);
    nFilterHeight : _UDINT(1);
    hrPrev : _HRESULT(S_OK);
	hresult : _HRESULT(S_OK);
END_VAR

METHOD PUBLIC  Clone : I_Node
VAR
	pNode : POINTER TO Node_F_VN_GaussianFilter;
END_VAR
pNode := __NEW(Node_F_VN_GaussianFilter);
Clone := pNode^;
END_METHOD

METHOD FB_init : BOOL
VAR_INPUT
	bInitRetains : BOOL; // if TRUE, the retain variables are initialized (warm start / cold start)
	bInCopyCode : BOOL;  // if TRUE, the instance afterwards gets moved into the copy code (online change)
END_VAR
AddInput('ipSrcImage', ipSrcImage);
AddParameter('nFilterWidth', nFilterWidth);
AddParameter('nFilterHeight', nFilterHeight);
AddInput('hrPrev', hrPrev);
AddOutput('ipDestImage', ipDestImage);
AddOutput('hresult',hresult);
END_METHOD

METHOD PROTECTED OnExecute
hresult.Value := F_VN_GaussianFilter(
	ipSrcImage:= ipSrcImage.Value, 
	ipDestImage:= ipDestImage.Value, 
	nFilterWidth:= nFilterWidth.Value, 
	nFilterHeight:= nFilterHeight.Value, 
	hrPrev:= hrPrev.Value);
END_METHOD

METHOD PUBLIC PreExecutionCheck
VAR_INPUT
	Check : I_PreExecutionChecks;
END_VAR
Check.IsTrue(ipSrcImage.IsValid, 'ipSrcImage must contain an image');
Check.IsTrue(nFilterWidth.IsOdd, 'nFilterWidth must be an odd number');
Check.IsTrue(nFilterHeight.IsOdd, 'nFilterHeight must be an odd number');
END_METHOD

END_FUNCTION_BLOCK

// ---- Nodes/Image Filtering/Node_F_VN_LaplacianFilter.TcPOU
{attribute 'linkalways'} 
{attribute 'no_explicit_call' := 'This FB is a CLASS and must be accessed using methods or properties'}
{attribute 'enable_dynamic_creation'}
FUNCTION_BLOCK Node_F_VN_LaplacianFilter EXTENDS VisionNode
VAR
	ipSrcImage : _ITcVnImage;
    ipDestImage : _ITcVnImage;
    eDestDepth : _ETcVnElementType(ETcVnElementType.TCVN_ET_SAME_AS_SOURCE);
    hrPrev : _HRESULT(S_OK);
	hresult : _HRESULT(S_OK);
END_VAR

METHOD PUBLIC  Clone : I_Node
VAR
	pNode : POINTER TO Node_F_VN_LaplacianFilter;
END_VAR
pNode := __NEW(Node_F_VN_LaplacianFilter);
Clone := pNode^;
END_METHOD

METHOD FB_init : BOOL
VAR_INPUT
	bInitRetains : BOOL; // if TRUE, the retain variables are initialized (warm start / cold start)
	bInCopyCode : BOOL;  // if TRUE, the instance afterwards gets moved into the copy code (online change)
END_VAR
AddInput('ipSrcImage', ipSrcImage);
AddParameter('eDestDepth', eDestDepth);
AddInput('hrPrev', hrPrev);
AddOutput('ipDestImage', ipDestImage);
AddOutput('hresult',hresult);
END_METHOD

METHOD PROTECTED OnExecute
hresult.Value := F_VN_LaplacianFilter(
	ipSrcImage := ipSrcImage.Value, 
	ipDestImage := ipDestImage.Value, 
	eDestDepth := eDestDepth.Value, 
	hrPrev := hrPrev.Value);
END_METHOD

METHOD PUBLIC PreExecutionCheck
VAR_INPUT
	Check : I_PreExecutionChecks;
END_VAR
VAR
	compatibleElementTypes_USINT : ARRAY [0..0] OF ETcVnElementType := [
		ETcVnElementType.TCVN_ET_USINT];
	
	compatibleElementTypes_UINT : ARRAY [0..1] OF ETcVnElementType := [
		ETcVnElementType.TCVN_ET_USINT,
		ETcVnElementType.TCVN_ET_UINT];
	
	compatibleElementTypes_INT : ARRAY [0..1] OF ETcVnElementType := [
		ETcVnElementType.TCVN_ET_USINT,
		ETcVnElementType.TCVN_ET_INT];
	
	compatibleElementTypes_REAL : ARRAY [0..3] OF ETcVnElementType := [
		ETcVnElementType.TCVN_ET_USINT,
		ETcVnElementType.TCVN_ET_UINT,
		ETcVnElementType.TCVN_ET_INT,
		ETcVnElementType.TCVN_ET_REAL];
	
	compatibleElementTypes_LREAL : ARRAY [0..3] OF ETcVnElementType := [
		ETcVnElementType.TCVN_ET_USINT,
		ETcVnElementType.TCVN_ET_UINT,
		ETcVnElementType.TCVN_ET_INT,
		ETcVnElementType.TCVN_ET_LREAL];
END_VAR
Check.IsTrue(ipSrcImage.IsValid, 'ipSrcImage must contain an image');

//The input image ipSrcImage may be in any available format, except for the data types SINT and DINT, which are generally not supported.

//Only the same or a larger data type than that of the input image can be used as the result depth, otherwise data would be lost.
//For example, a UINT cannot be converted to a USINT. 
//Furthermore, there are two restrictions, so that a UINT cannot be converted into an INT and a REAL cannot be converted into an LREAL.

CASE eDestDepth.Value OF
	ETcVnElementType.TCVN_ET_SINT,
    ETcVnElementType.TCVN_ET_DINT:
	    Check.Fail('ipSrcImage has unsupported pixel depth');
		RETURN;
END_CASE

CASE eDestDepth.Value OF
    ETcVnElementType.TCVN_ET_SINT,
    ETcVnElementType.TCVN_ET_DINT:
	    Check.Fail('ipSrcImage has unsupported pixel depth');
		RETURN;
        
	ETcVnElementType.TCVN_ET_USINT:
        Check.IsTrue(ImageHasCompatibleElementType(ipSrcImage.Value, compatibleElementTypes_USINT), 'ipSrcImage has incompatible pixel depth');
	
	ETcVnElementType.TCVN_ET_UINT:
	    Check.IsTrue(ImageHasCompatibleElementType(ipSrcImage.Value, compatibleElementTypes_UINT), 'ipSrcImage has incompatible pixel depth');
		
	ETcVnElementType.TCVN_ET_INT:
	    Check.IsTrue(ImageHasCompatibleElementType(ipSrcImage.Value, compatibleElementTypes_INT), 'ipSrcImage has incompatible pixel depth');
	
	ETcVnElementType.TCVN_ET_REAL:
	    Check.IsTrue(ImageHasCompatibleElementType(ipSrcImage.Value, compatibleElementTypes_REAL), 'ipSrcImage has incompatible pixel depth');
	
	ETcVnElementType.TCVN_ET_LREAL:
	    Check.IsTrue(ImageHasCompatibleElementType(ipSrcImage.Value, compatibleElementTypes_LREAL), 'ipSrcImage has incompatible pixel depth');
END_CASE
END_METHOD

END_FUNCTION_BLOCK

// ---- Nodes/Image Filtering/Node_F_VN_LocalMinima.TcPOU
{attribute 'linkalways'} 
{attribute 'no_explicit_call' := 'This FB is a CLASS and must be accessed using methods or properties'}
{attribute 'enable_dynamic_creation'}
FUNCTION_BLOCK Node_F_VN_LocalMinima EXTENDS VisionNode
VAR
    ipSrcImage : _ITcVnImage;
    ipDestImage : _ITcVnImage;
    hrPrev : _HRESULT(S_OK);
	hresult : _HRESULT(S_OK);
END_VAR

METHOD PUBLIC  Clone : I_Node
VAR
	pNode : POINTER TO Node_F_VN_LocalMinima;
END_VAR
pNode := __NEW(Node_F_VN_LocalMinima);
Clone := pNode^;
END_METHOD

METHOD FB_init : BOOL
VAR_INPUT
	bInitRetains : BOOL; // if TRUE, the retain variables are initialized (warm start / cold start)
	bInCopyCode : BOOL;  // if TRUE, the instance afterwards gets moved into the copy code (online change)
END_VAR
AddInput('ipSrcImage', ipSrcImage);
AddInput('hrPrev', hrPrev);
AddOutput('ipDestImage', ipDestImage);
AddOutput('hresult',hresult);
END_METHOD

METHOD PROTECTED OnExecute
hresult.Value := F_VN_LocalMinima(
    ipSrcImage := ipSrcImage.Value,
	ipDestImage := ipDestImage.Value,
	hrPrev:= hrPrev.Value);
END_METHOD

METHOD PUBLIC PreExecutionCheck
VAR_INPUT
	Check : I_PreExecutionChecks;
END_VAR
Check.IsTrue(ipSrcImage.IsValid, 'ipSrcImage must contain an image');
Check.IsTrue(ipSrcImage.HasChannelCount(1), 'ipSrcImage must have 1 channel');

Check.IsTrue((ipSrcImage.IsPixelDepth(8)  OR
              ipSrcImage.IsPixelDepth(16)), 'ipSrcImage must have 8 or 16 bit pixel depth');
END_METHOD

END_FUNCTION_BLOCK

// ---- Nodes/Image Filtering/Node_F_VN_VarianceFilterExp.TcPOU
{attribute 'linkalways'} 
{attribute 'no_explicit_call' := 'This FB is a CLASS and must be accessed using methods or properties'}
{attribute 'enable_dynamic_creation'}
FUNCTION_BLOCK Node_F_VN_VarianceFilterExp EXTENDS VisionNode
VAR
    ipSrcImage : _ITcVnImage;
    ipDestImage : _ITcVnImage;
    nKernelSize : _UDINT(0);
    fScale : _LREAL(1.0);
    eBorderType : _ETcVnBorderInterpolationMethod(ETcVnBorderInterpolationMethod.TCVN_BIM_DEFAULT);
    hrPrev : _HRESULT(S_OK);
	hresult : _HRESULT(S_OK);
END_VAR

METHOD PUBLIC  Clone : I_Node
VAR
	pNode : POINTER TO Node_F_VN_VarianceFilterExp;
END_VAR
pNode := __NEW(Node_F_VN_VarianceFilterExp);
Clone := pNode^;
END_METHOD

METHOD FB_init : BOOL
VAR_INPUT
	bInitRetains : BOOL; // if TRUE, the retain variables are initialized (warm start / cold start)
	bInCopyCode : BOOL;  // if TRUE, the instance afterwards gets moved into the copy code (online change)
END_VAR
AddInput('ipSrcImage', ipSrcImage);
AddParameter('nKernelSize', nKernelSize);
AddParameter('fScale', fScale);
AddParameter('eBorderType', eBorderType);
AddInput('hrPrev', hrPrev);
AddOutput('ipDestImage', ipDestImage);
AddOutput('hresult',hresult);
END_METHOD

METHOD PROTECTED OnExecute
hresult.Value := F_VN_VarianceFilterExp(
    ipSrcImage := ipSrcImage.Value,
	ipDestImage := ipDestImage.Value,
    nKernelSize := nKernelSize.Value,
    fScale := fScale.Value,
    eBorderType := eBorderType.Value,
	hrPrev:= hrPrev.Value);
END_METHOD

METHOD PUBLIC PreExecutionCheck
VAR_INPUT
	Check : I_PreExecutionChecks;
END_VAR
Check.IsTrue(ipSrcImage.IsValid, 'ipSrcImage must contain an image');
Check.IsTrue(ipSrcImage.HasChannelCount(1), 'ipSrcImage must have 1 channel');
Check.IsTrue(ipSrcImage.IsPixelDepth(8), 'ipSrcImage must have 8 bit pixel depth');
END_METHOD

END_FUNCTION_BLOCK

// ---- Nodes/Image Segmentation/Node_F_VN_AdaptiveThresholdExp.TcPOU
{attribute 'linkalways'} 
{attribute 'no_explicit_call' := 'This FB is a CLASS and must be accessed using methods or properties'}
{attribute 'enable_dynamic_creation'}
FUNCTION_BLOCK Node_F_VN_AdaptiveThresholdExp EXTENDS VisionNode
VAR
	ipSrcImage : _ITcVnImage;
    ipDestImage : _ITcVnImage;
    fMaxValue : _LREAL(0.0);
    eAdaptiveMethod : _ETcVnAdaptiveThresholdMethod(ETcVnAdaptiveThresholdMethod.TCVN_ATM_MEAN);
    eThresholdType : _ETcVnThresholdType(ETcVnThresholdType.TCVN_TT_BINARY);
    nBlockSize : _UDINT(3);
    fConstant : _LREAL(0.0);
    hrPrev : _HRESULT(S_OK);
	hresult : _HRESULT(S_OK);
END_VAR

METHOD PUBLIC  Clone : I_Node
VAR
	pNode : POINTER TO Node_F_VN_AdaptiveThresholdExp;
END_VAR
pNode := __NEW(Node_F_VN_AdaptiveThresholdExp);
Clone := pNode^;
END_METHOD

METHOD FB_init : BOOL
VAR_INPUT
	bInitRetains : BOOL; // if TRUE, the retain variables are initialized (warm start / cold start)
	bInCopyCode : BOOL;  // if TRUE, the instance afterwards gets moved into the copy code (online change)
END_VAR
AddInput('ipSrcImage', ipSrcImage);
AddParameter('fMaxValue', fMaxValue);
AddParameter('eAdaptiveMethod', eAdaptiveMethod);
AddParameter('eThresholdType', eThresholdType);
AddParameter('nBlockSize', nBlockSize);
AddParameter('fConstant', fConstant);
AddInput('hrPrev', hrPrev);
AddOutput('ipDestImage', ipDestImage);
AddOutput('hresult', hresult);
END_METHOD

METHOD PROTECTED OnExecute
hresult.Value := F_VN_AdaptiveThresholdExp(
	ipSrcImage := ipSrcImage.Value,
	ipDestImage := ipDestImage.Value,
    fMaxValue := fMaxValue.Value,
    eAdaptiveMethod := eAdaptiveMethod.Value,
    eThresholdType := eThresholdType.Value,
    nBlockSize := nBlockSize.Value,
    fConstant := fConstant.Value,
	hrPrev := hrPrev.Value);
END_METHOD

